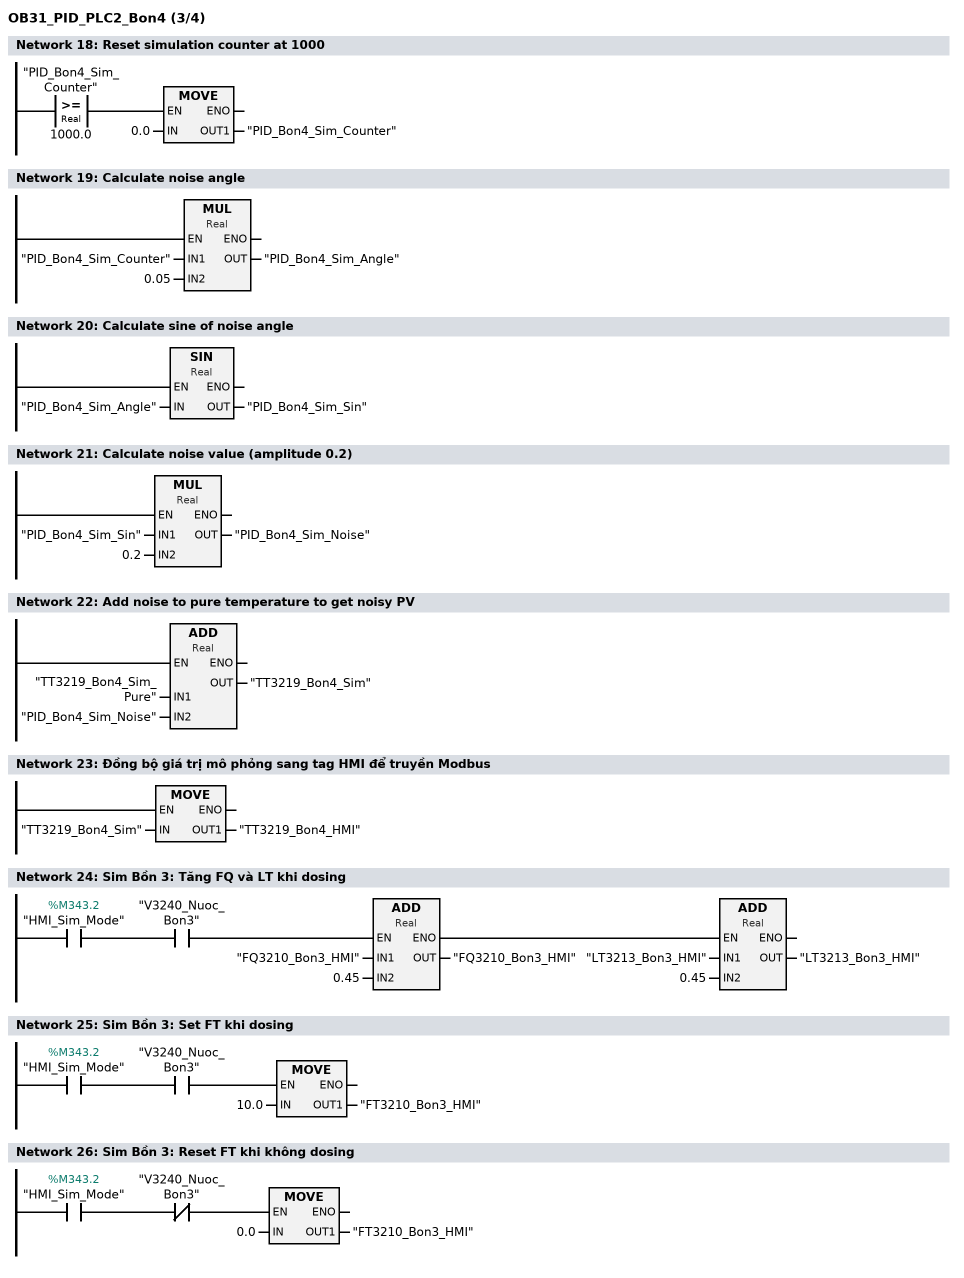
   RUNG wire#powerrail
      { S7_Templates := "SrcType := Real" } GE_Contact(in1 := "PID_Bon4_Sim_Counter", in2 := 1000.0)
      { S7_GenerateENO := "TRUE" } Move(in := 0.0, out1 => "PID_Bon4_Sim_Counter")
   END_RUNG
   // the same network as SCL:
   IF "PID_Bon4_Sim_Counter" >= 1000.0 THEN "PID_Bon4_Sim_Counter" := 0.0; END_IF;
END_REGION

REGION Network 19: Calculate noise angle
   RUNG wire#powerrail
      { S7_Templates := "SrcType := Real"; S7_GenerateENO := "TRUE" } Mul(in1 := "PID_Bon4_Sim_Counter", in2 := 0.05, out => "PID_Bon4_Sim_Angle")
   END_RUNG
   // the same network as SCL:
   "PID_Bon4_Sim_Angle" := "PID_Bon4_Sim_Counter" * 0.05;
END_REGION

REGION Network 20: Calculate sine of noise angle
   "PID_Bon4_Sim_Sin" := SIN("PID_Bon4_Sim_Angle");
END_REGION

REGION Network 21: Calculate noise value (amplitude 0.2)
   RUNG wire#powerrail
      { S7_Templates := "SrcType := Real"; S7_GenerateENO := "TRUE" } Mul(in1 := "PID_Bon4_Sim_Sin", in2 := 0.2, out => "PID_Bon4_Sim_Noise")
   END_RUNG
   // the same network as SCL:
   "PID_Bon4_Sim_Noise" := "PID_Bon4_Sim_Sin" * 0.2;
END_REGION

REGION Network 22: Add noise to pure temperature to get noisy PV
   RUNG wire#powerrail
      { S7_Templates := "SrcType := Real"; S7_GenerateENO := "TRUE" } Add(in1 := "TT3219_Bon4_Sim_Pure", in2 := "PID_Bon4_Sim_Noise", out => "TT3219_Bon4_Sim")
   END_RUNG
   // the same network as SCL:
   "TT3219_Bon4_Sim" := "TT3219_Bon4_Sim_Pure" + "PID_Bon4_Sim_Noise";
END_REGION

REGION Network 23: Đồng bộ giá trị mô phỏng sang tag HMI để truyền Modbus
   RUNG wire#powerrail
      { S7_GenerateENO := "TRUE" } Move(in := "TT3219_Bon4_Sim", out1 => "TT3219_Bon4_HMI")
   END_RUNG
   // the same network as SCL:
   "TT3219_Bon4_HMI" := "TT3219_Bon4_Sim";
END_REGION

REGION Network 24: Sim Bồn 3: Tăng FQ và LT khi dosing
   RUNG wire#powerrail
      Contact( "HMI_Sim_Mode" )
      Contact( "V3240_Nuoc_Bon3" )
      { S7_Templates := "SrcType := Real"; S7_GenerateENO := "TRUE" } Add(in1 := "FQ3210_Bon3_HMI", in2 := 0.45, out => "FQ3210_Bon3_HMI")
      { S7_Templates := "SrcType := Real"; S7_GenerateENO := "TRUE" } Add(in1 := "LT3213_Bon3_HMI", in2 := 0.45, out => "LT3213_Bon3_HMI")
   END_RUNG
   // the same network as SCL:
   // ENO of a box is taken as its EN; it also drops when the box reports an error
   IF "HMI_Sim_Mode" AND "V3240_Nuoc_Bon3" THEN
       "FQ3210_Bon3_HMI" := "FQ3210_Bon3_HMI" + 0.45;
       "LT3213_Bon3_HMI" := "LT3213_Bon3_HMI" + 0.45;
   END_IF;
END_REGION

REGION Network 25: Sim Bồn 3: Set FT khi dosing
   RUNG wire#powerrail
      Contact( "HMI_Sim_Mode" )
      Contact( "V3240_Nuoc_Bon3" )
      { S7_GenerateENO := "TRUE" } Move(in := 10.0, out1 => "FT3210_Bon3_HMI")
   END_RUNG
   // the same network as SCL:
   IF "HMI_Sim_Mode" AND "V3240_Nuoc_Bon3" THEN "FT3210_Bon3_HMI" := 10.0; END_IF;
END_REGION

REGION Network 26: Sim Bồn 3: Reset FT khi không dosing
   RUNG wire#powerrail
      Contact( "HMI_Sim_Mode" )
      I_Contact( "V3240_Nuoc_Bon3" )
      { S7_GenerateENO := "TRUE" } Move(in := 0.0, out1 => "FT3210_Bon3_HMI")
   END_RUNG
   // the same network as SCL:
   IF "HMI_Sim_Mode" AND NOT "V3240_Nuoc_Bon3" THEN "FT3210_Bon3_HMI" := 0.0; END_IF;
END_REGION

REGION Network 27: Sim Bồn 3: Giảm LT khi xả đáy
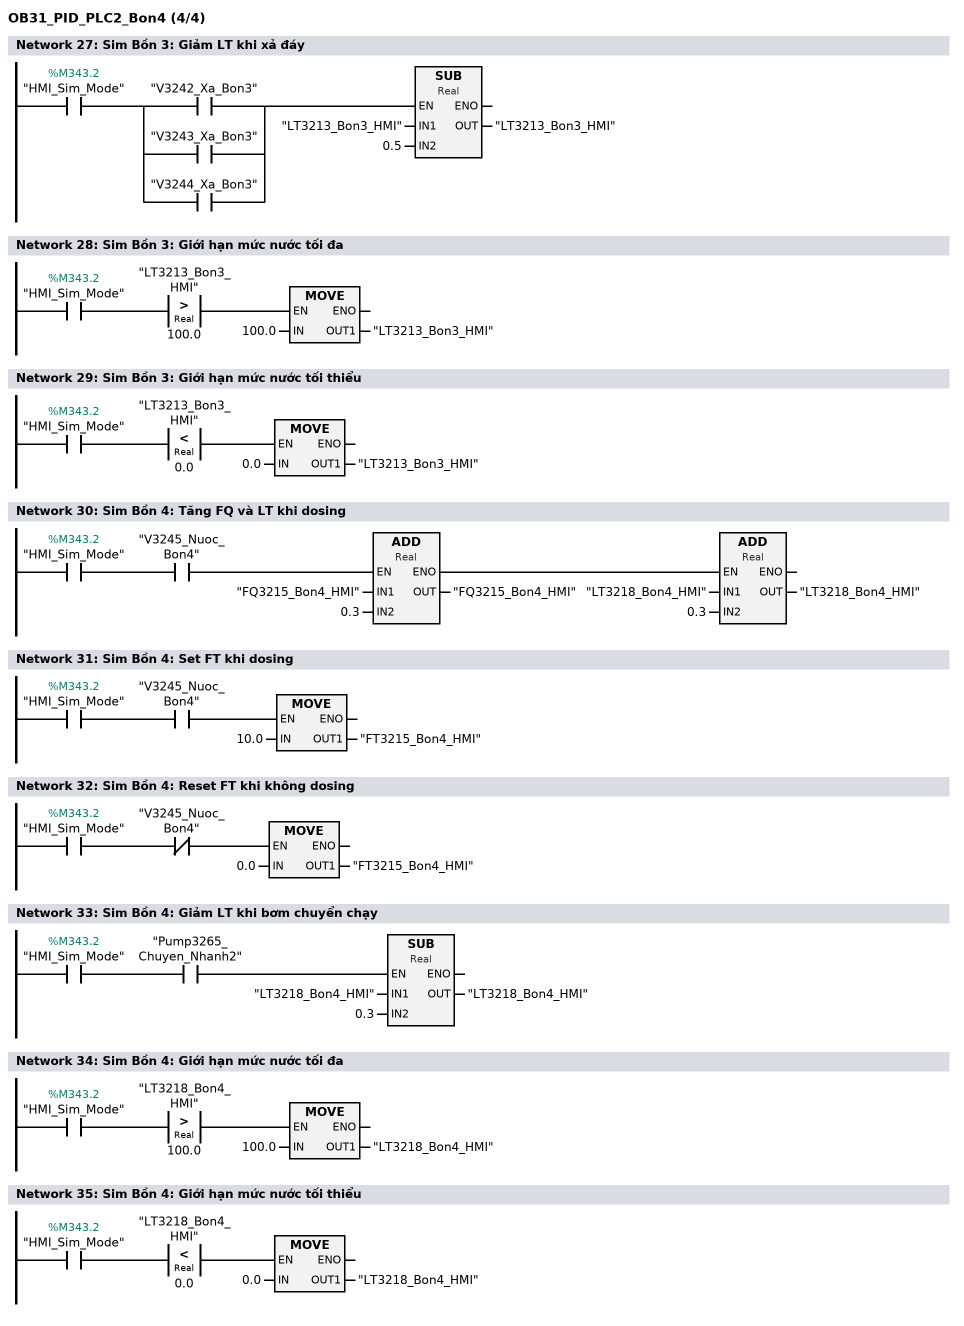
   RUNG wire#powerrail
      Contact( "HMI_Sim_Mode" )
      wire#w1
      Contact( "V3242_Xa_Bon3" )
      wire#w2
      { S7_Templates := "SrcType := Real"; S7_GenerateENO := "TRUE" } Sub(in1 := "LT3213_Bon3_HMI", in2 := 0.5, out => "LT3213_Bon3_HMI")
   END_RUNG
   RUNG wire#w1
      Contact( "V3243_Xa_Bon3" )
   END_RUNG wire#w2
   RUNG wire#w1
      Contact( "V3244_Xa_Bon3" )
   END_RUNG wire#w2
   // the same network as SCL:
   IF "HMI_Sim_Mode" AND ("V3242_Xa_Bon3" OR "V3243_Xa_Bon3" OR "V3244_Xa_Bon3") THEN
       "LT3213_Bon3_HMI" := "LT3213_Bon3_HMI" - 0.5;
   END_IF;
END_REGION

REGION Network 28: Sim Bồn 3: Giới hạn mức nước tối đa
   RUNG wire#powerrail
      Contact( "HMI_Sim_Mode" )
      { S7_Templates := "SrcType := Real" } GT_Contact(in1 := "LT3213_Bon3_HMI", in2 := 100.0)
      { S7_GenerateENO := "TRUE" } Move(in := 100.0, out1 => "LT3213_Bon3_HMI")
   END_RUNG
   // the same network as SCL:
   IF "HMI_Sim_Mode" AND ("LT3213_Bon3_HMI" > 100.0) THEN "LT3213_Bon3_HMI" := 100.0; END_IF;
END_REGION

REGION Network 29: Sim Bồn 3: Giới hạn mức nước tối thiểu
   RUNG wire#powerrail
      Contact( "HMI_Sim_Mode" )
      { S7_Templates := "SrcType := Real" } LT_Contact(in1 := "LT3213_Bon3_HMI", in2 := 0.0)
      { S7_GenerateENO := "TRUE" } Move(in := 0.0, out1 => "LT3213_Bon3_HMI")
   END_RUNG
   // the same network as SCL:
   IF "HMI_Sim_Mode" AND ("LT3213_Bon3_HMI" < 0.0) THEN "LT3213_Bon3_HMI" := 0.0; END_IF;
END_REGION

REGION Network 30: Sim Bồn 4: Tăng FQ và LT khi dosing
   RUNG wire#powerrail
      Contact( "HMI_Sim_Mode" )
      Contact( "V3245_Nuoc_Bon4" )
      { S7_Templates := "SrcType := Real"; S7_GenerateENO := "TRUE" } Add(in1 := "FQ3215_Bon4_HMI", in2 := 0.3, out => "FQ3215_Bon4_HMI")
      { S7_Templates := "SrcType := Real"; S7_GenerateENO := "TRUE" } Add(in1 := "LT3218_Bon4_HMI", in2 := 0.3, out => "LT3218_Bon4_HMI")
   END_RUNG
   // the same network as SCL:
   // ENO of a box is taken as its EN; it also drops when the box reports an error
   IF "HMI_Sim_Mode" AND "V3245_Nuoc_Bon4" THEN
       "FQ3215_Bon4_HMI" := "FQ3215_Bon4_HMI" + 0.3;
       "LT3218_Bon4_HMI" := "LT3218_Bon4_HMI" + 0.3;
   END_IF;
END_REGION

REGION Network 31: Sim Bồn 4: Set FT khi dosing
   RUNG wire#powerrail
      Contact( "HMI_Sim_Mode" )
      Contact( "V3245_Nuoc_Bon4" )
      { S7_GenerateENO := "TRUE" } Move(in := 10.0, out1 => "FT3215_Bon4_HMI")
   END_RUNG
   // the same network as SCL:
   IF "HMI_Sim_Mode" AND "V3245_Nuoc_Bon4" THEN "FT3215_Bon4_HMI" := 10.0; END_IF;
END_REGION

REGION Network 32: Sim Bồn 4: Reset FT khi không dosing
   RUNG wire#powerrail
      Contact( "HMI_Sim_Mode" )
      I_Contact( "V3245_Nuoc_Bon4" )
      { S7_GenerateENO := "TRUE" } Move(in := 0.0, out1 => "FT3215_Bon4_HMI")
   END_RUNG
   // the same network as SCL:
   IF "HMI_Sim_Mode" AND NOT "V3245_Nuoc_Bon4" THEN "FT3215_Bon4_HMI" := 0.0; END_IF;
END_REGION

REGION Network 33: Sim Bồn 4: Giảm LT khi bơm chuyển chạy
   RUNG wire#powerrail
      Contact( "HMI_Sim_Mode" )
      Contact( "Pump3265_Chuyen_Nhanh2" )
      { S7_Templates := "SrcType := Real"; S7_GenerateENO := "TRUE" } Sub(in1 := "LT3218_Bon4_HMI", in2 := 0.3, out => "LT3218_Bon4_HMI")
   END_RUNG
   // the same network as SCL:
   IF "HMI_Sim_Mode" AND "Pump3265_Chuyen_Nhanh2" THEN "LT3218_Bon4_HMI" := "LT3218_Bon4_HMI" - 0.3; END_IF;
END_REGION

REGION Network 34: Sim Bồn 4: Giới hạn mức nước tối đa
   RUNG wire#powerrail
      Contact( "HMI_Sim_Mode" )
      { S7_Templates := "SrcType := Real" } GT_Contact(in1 := "LT3218_Bon4_HMI", in2 := 100.0)
      { S7_GenerateENO := "TRUE" } Move(in := 100.0, out1 => "LT3218_Bon4_HMI")
   END_RUNG
   // the same network as SCL:
   IF "HMI_Sim_Mode" AND ("LT3218_Bon4_HMI" > 100.0) THEN "LT3218_Bon4_HMI" := 100.0; END_IF;
END_REGION

REGION Network 35: Sim Bồn 4: Giới hạn mức nước tối thiểu
   RUNG wire#powerrail
      Contact( "HMI_Sim_Mode" )
      { S7_Templates := "SrcType := Real" } LT_Contact(in1 := "LT3218_Bon4_HMI", in2 := 0.0)
      { S7_GenerateENO := "TRUE" } Move(in := 0.0, out1 => "LT3218_Bon4_HMI")
   END_RUNG
   // the same network as SCL:
   IF "HMI_Sim_Mode" AND ("LT3218_Bon4_HMI" < 0.0) THEN "LT3218_Bon4_HMI" := 0.0; END_IF;
END_REGION
END_ORGANIZATION_BLOCK

FUNCTION "FC_HMI_Mirror_PLC2" : Void   // FC41, LAD
{ S7_Optimized_Access := 'TRUE' }
VERSION : 0.1
// stored: AutoNumber true, IsIECCheckEnabled false, SetENOAutomatically false, UDAEnableTagReadback false
BEGIN

REGION Network 1: Mirror V3240_Nuoc_Bon3
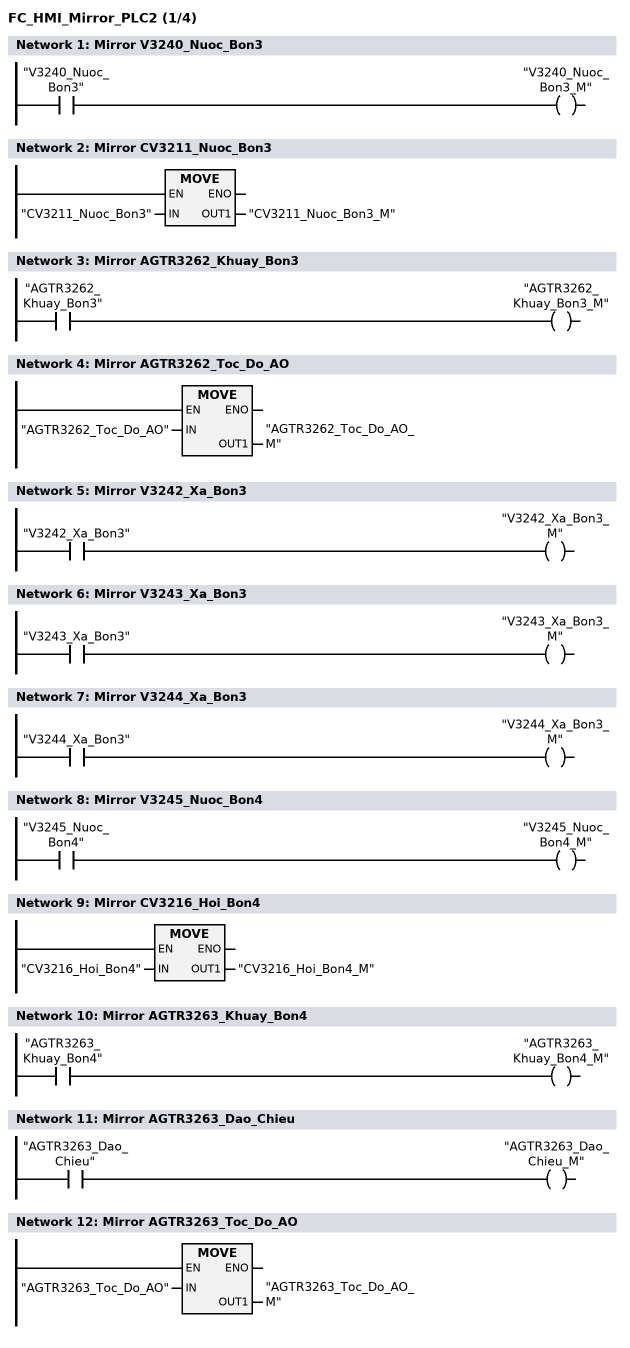
   RUNG wire#powerrail
      Contact( "V3240_Nuoc_Bon3" )
      Coil( "V3240_Nuoc_Bon3_M" )
   END_RUNG
   // the same network as SCL:
   "V3240_Nuoc_Bon3_M" := "V3240_Nuoc_Bon3";
END_REGION

REGION Network 2: Mirror CV3211_Nuoc_Bon3
   RUNG wire#powerrail
      { S7_GenerateENO := "TRUE" } Move(in := "CV3211_Nuoc_Bon3", out1 => "CV3211_Nuoc_Bon3_M")
   END_RUNG
   // the same network as SCL:
   "CV3211_Nuoc_Bon3_M" := "CV3211_Nuoc_Bon3";
END_REGION

REGION Network 3: Mirror AGTR3262_Khuay_Bon3
   RUNG wire#powerrail
      Contact( "AGTR3262_Khuay_Bon3" )
      Coil( "AGTR3262_Khuay_Bon3_M" )
   END_RUNG
   // the same network as SCL:
   "AGTR3262_Khuay_Bon3_M" := "AGTR3262_Khuay_Bon3";
END_REGION

REGION Network 4: Mirror AGTR3262_Toc_Do_AO
   RUNG wire#powerrail
      { S7_GenerateENO := "TRUE" } Move(in := "AGTR3262_Toc_Do_AO", out1 => "AGTR3262_Toc_Do_AO_M")
   END_RUNG
   // the same network as SCL:
   "AGTR3262_Toc_Do_AO_M" := "AGTR3262_Toc_Do_AO";
END_REGION

REGION Network 5: Mirror V3242_Xa_Bon3
   RUNG wire#powerrail
      Contact( "V3242_Xa_Bon3" )
      Coil( "V3242_Xa_Bon3_M" )
   END_RUNG
   // the same network as SCL:
   "V3242_Xa_Bon3_M" := "V3242_Xa_Bon3";
END_REGION

REGION Network 6: Mirror V3243_Xa_Bon3
   RUNG wire#powerrail
      Contact( "V3243_Xa_Bon3" )
      Coil( "V3243_Xa_Bon3_M" )
   END_RUNG
   // the same network as SCL:
   "V3243_Xa_Bon3_M" := "V3243_Xa_Bon3";
END_REGION

REGION Network 7: Mirror V3244_Xa_Bon3
   RUNG wire#powerrail
      Contact( "V3244_Xa_Bon3" )
      Coil( "V3244_Xa_Bon3_M" )
   END_RUNG
   // the same network as SCL:
   "V3244_Xa_Bon3_M" := "V3244_Xa_Bon3";
END_REGION

REGION Network 8: Mirror V3245_Nuoc_Bon4
   RUNG wire#powerrail
      Contact( "V3245_Nuoc_Bon4" )
      Coil( "V3245_Nuoc_Bon4_M" )
   END_RUNG
   // the same network as SCL:
   "V3245_Nuoc_Bon4_M" := "V3245_Nuoc_Bon4";
END_REGION

REGION Network 9: Mirror CV3216_Hoi_Bon4
   RUNG wire#powerrail
      { S7_GenerateENO := "TRUE" } Move(in := "CV3216_Hoi_Bon4", out1 => "CV3216_Hoi_Bon4_M")
   END_RUNG
   // the same network as SCL:
   "CV3216_Hoi_Bon4_M" := "CV3216_Hoi_Bon4";
END_REGION

REGION Network 10: Mirror AGTR3263_Khuay_Bon4
   RUNG wire#powerrail
      Contact( "AGTR3263_Khuay_Bon4" )
      Coil( "AGTR3263_Khuay_Bon4_M" )
   END_RUNG
   // the same network as SCL:
   "AGTR3263_Khuay_Bon4_M" := "AGTR3263_Khuay_Bon4";
END_REGION

REGION Network 11: Mirror AGTR3263_Dao_Chieu
   RUNG wire#powerrail
      Contact( "AGTR3263_Dao_Chieu" )
      Coil( "AGTR3263_Dao_Chieu_M" )
   END_RUNG
   // the same network as SCL:
   "AGTR3263_Dao_Chieu_M" := "AGTR3263_Dao_Chieu";
END_REGION

REGION Network 12: Mirror AGTR3263_Toc_Do_AO
   RUNG wire#powerrail
      { S7_GenerateENO := "TRUE" } Move(in := "AGTR3263_Toc_Do_AO", out1 => "AGTR3263_Toc_Do_AO_M")
   END_RUNG
   // the same network as SCL:
   "AGTR3263_Toc_Do_AO_M" := "AGTR3263_Toc_Do_AO";
END_REGION

REGION Network 13: Mirror V3247_Xa_Bon4
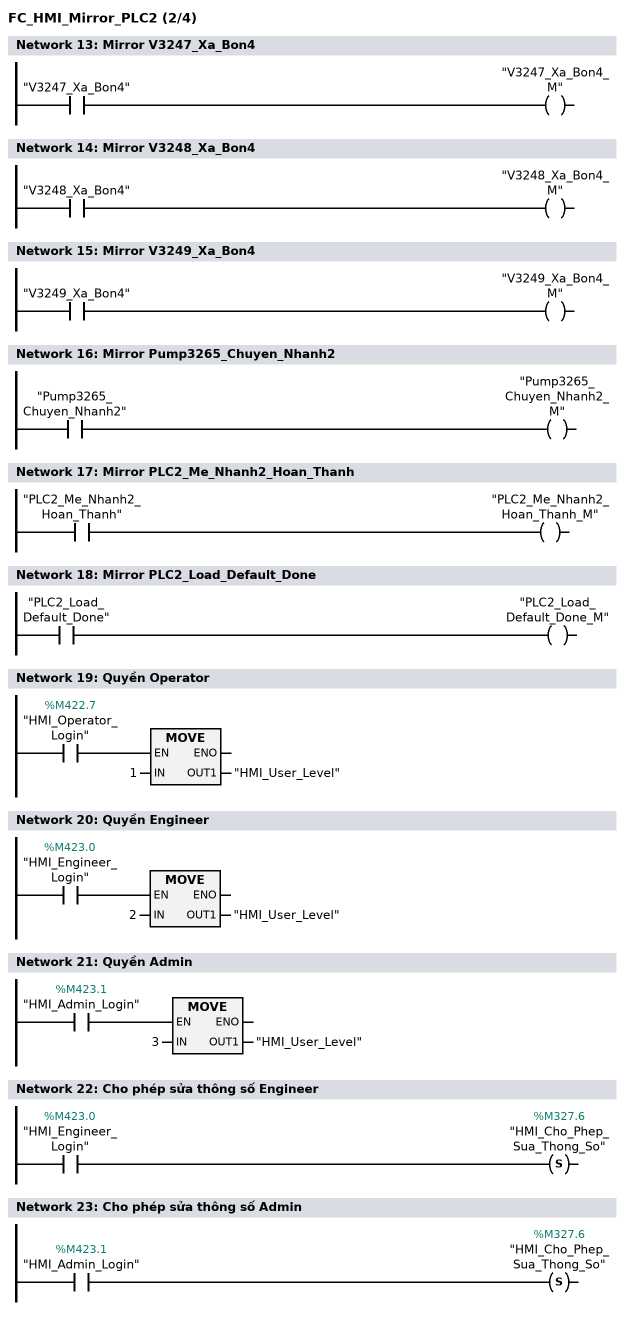
   RUNG wire#powerrail
      Contact( "V3247_Xa_Bon4" )
      Coil( "V3247_Xa_Bon4_M" )
   END_RUNG
   // the same network as SCL:
   "V3247_Xa_Bon4_M" := "V3247_Xa_Bon4";
END_REGION

REGION Network 14: Mirror V3248_Xa_Bon4
   RUNG wire#powerrail
      Contact( "V3248_Xa_Bon4" )
      Coil( "V3248_Xa_Bon4_M" )
   END_RUNG
   // the same network as SCL:
   "V3248_Xa_Bon4_M" := "V3248_Xa_Bon4";
END_REGION

REGION Network 15: Mirror V3249_Xa_Bon4
   RUNG wire#powerrail
      Contact( "V3249_Xa_Bon4" )
      Coil( "V3249_Xa_Bon4_M" )
   END_RUNG
   // the same network as SCL:
   "V3249_Xa_Bon4_M" := "V3249_Xa_Bon4";
END_REGION

REGION Network 16: Mirror Pump3265_Chuyen_Nhanh2
   RUNG wire#powerrail
      Contact( "Pump3265_Chuyen_Nhanh2" )
      Coil( "Pump3265_Chuyen_Nhanh2_M" )
   END_RUNG
   // the same network as SCL:
   "Pump3265_Chuyen_Nhanh2_M" := "Pump3265_Chuyen_Nhanh2";
END_REGION

REGION Network 17: Mirror PLC2_Me_Nhanh2_Hoan_Thanh
   RUNG wire#powerrail
      Contact( "PLC2_Me_Nhanh2_Hoan_Thanh" )
      Coil( "PLC2_Me_Nhanh2_Hoan_Thanh_M" )
   END_RUNG
   // the same network as SCL:
   "PLC2_Me_Nhanh2_Hoan_Thanh_M" := "PLC2_Me_Nhanh2_Hoan_Thanh";
END_REGION

REGION Network 18: Mirror PLC2_Load_Default_Done
   RUNG wire#powerrail
      Contact( "PLC2_Load_Default_Done" )
      Coil( "PLC2_Load_Default_Done_M" )
   END_RUNG
   // the same network as SCL:
   "PLC2_Load_Default_Done_M" := "PLC2_Load_Default_Done";
END_REGION

REGION Network 19: Quyền Operator
   RUNG wire#powerrail
      Contact( "HMI_Operator_Login" )
      { S7_GenerateENO := "TRUE" } Move(in := 1, out1 => "HMI_User_Level")
   END_RUNG
   // the same network as SCL:
   IF "HMI_Operator_Login" THEN "HMI_User_Level" := 1; END_IF;
END_REGION

REGION Network 20: Quyền Engineer
   RUNG wire#powerrail
      Contact( "HMI_Engineer_Login" )
      { S7_GenerateENO := "TRUE" } Move(in := 2, out1 => "HMI_User_Level")
   END_RUNG
   // the same network as SCL:
   IF "HMI_Engineer_Login" THEN "HMI_User_Level" := 2; END_IF;
END_REGION

REGION Network 21: Quyền Admin
   RUNG wire#powerrail
      Contact( "HMI_Admin_Login" )
      { S7_GenerateENO := "TRUE" } Move(in := 3, out1 => "HMI_User_Level")
   END_RUNG
   // the same network as SCL:
   IF "HMI_Admin_Login" THEN "HMI_User_Level" := 3; END_IF;
END_REGION

REGION Network 22: Cho phép sửa thông số Engineer
   RUNG wire#powerrail
      Contact( "HMI_Engineer_Login" )
      S_Coil( "HMI_Cho_Phep_Sua_Thong_So" )
   END_RUNG
   // the same network as SCL:
   IF "HMI_Engineer_Login" THEN "HMI_Cho_Phep_Sua_Thong_So" := TRUE; END_IF;
END_REGION

REGION Network 23: Cho phép sửa thông số Admin
   RUNG wire#powerrail
      Contact( "HMI_Admin_Login" )
      S_Coil( "HMI_Cho_Phep_Sua_Thong_So" )
   END_RUNG
   // the same network as SCL:
   IF "HMI_Admin_Login" THEN "HMI_Cho_Phep_Sua_Thong_So" := TRUE; END_IF;
END_REGION

REGION Network 24: Operator không được sửa thông số
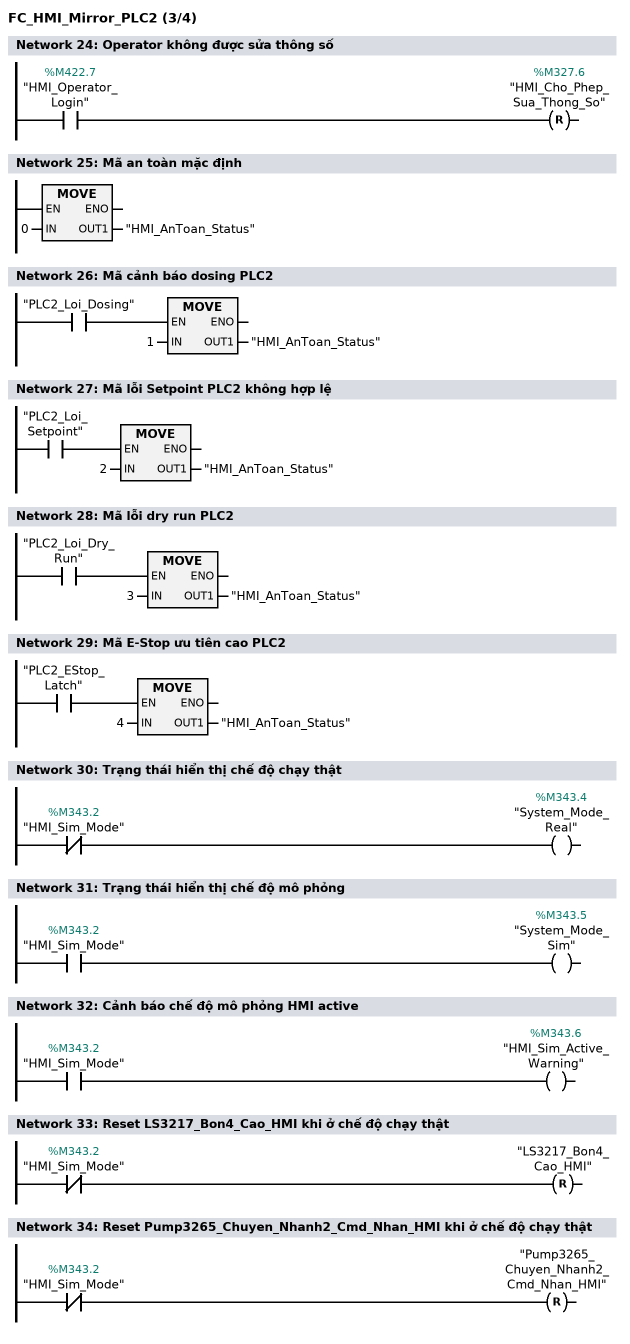
   RUNG wire#powerrail
      Contact( "HMI_Operator_Login" )
      R_Coil( "HMI_Cho_Phep_Sua_Thong_So" )
   END_RUNG
   // the same network as SCL:
   IF "HMI_Operator_Login" THEN "HMI_Cho_Phep_Sua_Thong_So" := FALSE; END_IF;
END_REGION

REGION Network 25: Mã an toàn mặc định
   RUNG wire#powerrail
      { S7_GenerateENO := "TRUE" } Move(in := 0, out1 => "HMI_AnToan_Status")
   END_RUNG
   // the same network as SCL:
   "HMI_AnToan_Status" := 0;
END_REGION

REGION Network 26: Mã cảnh báo dosing PLC2
   RUNG wire#powerrail
      Contact( "PLC2_Loi_Dosing" )
      { S7_GenerateENO := "TRUE" } Move(in := 1, out1 => "HMI_AnToan_Status")
   END_RUNG
   // the same network as SCL:
   IF "PLC2_Loi_Dosing" THEN "HMI_AnToan_Status" := 1; END_IF;
END_REGION

REGION Network 27: Mã lỗi Setpoint PLC2 không hợp lệ
   RUNG wire#powerrail
      Contact( "PLC2_Loi_Setpoint" )
      { S7_GenerateENO := "TRUE" } Move(in := 2, out1 => "HMI_AnToan_Status")
   END_RUNG
   // the same network as SCL:
   IF "PLC2_Loi_Setpoint" THEN "HMI_AnToan_Status" := 2; END_IF;
END_REGION

REGION Network 28: Mã lỗi dry run PLC2
   RUNG wire#powerrail
      Contact( "PLC2_Loi_Dry_Run" )
      { S7_GenerateENO := "TRUE" } Move(in := 3, out1 => "HMI_AnToan_Status")
   END_RUNG
   // the same network as SCL:
   IF "PLC2_Loi_Dry_Run" THEN "HMI_AnToan_Status" := 3; END_IF;
END_REGION

REGION Network 29: Mã E-Stop ưu tiên cao PLC2
   RUNG wire#powerrail
      Contact( "PLC2_EStop_Latch" )
      { S7_GenerateENO := "TRUE" } Move(in := 4, out1 => "HMI_AnToan_Status")
   END_RUNG
   // the same network as SCL:
   IF "PLC2_EStop_Latch" THEN "HMI_AnToan_Status" := 4; END_IF;
END_REGION

REGION Network 30: Trạng thái hiển thị chế độ chạy thật
   RUNG wire#powerrail
      I_Contact( "HMI_Sim_Mode" )
      Coil( "System_Mode_Real" )
   END_RUNG
   // the same network as SCL:
   "System_Mode_Real" := NOT "HMI_Sim_Mode";
END_REGION

REGION Network 31: Trạng thái hiển thị chế độ mô phỏng
   RUNG wire#powerrail
      Contact( "HMI_Sim_Mode" )
      Coil( "System_Mode_Sim" )
   END_RUNG
   // the same network as SCL:
   "System_Mode_Sim" := "HMI_Sim_Mode";
END_REGION

REGION Network 32: Cảnh báo chế độ mô phỏng HMI active
   RUNG wire#powerrail
      Contact( "HMI_Sim_Mode" )
      Coil( "HMI_Sim_Active_Warning" )
   END_RUNG
   // the same network as SCL:
   "HMI_Sim_Active_Warning" := "HMI_Sim_Mode";
END_REGION

REGION Network 33: Reset LS3217_Bon4_Cao_HMI khi ở chế độ chạy thật
   RUNG wire#powerrail
      I_Contact( "HMI_Sim_Mode" )
      R_Coil( "LS3217_Bon4_Cao_HMI" )
   END_RUNG
   // the same network as SCL:
   IF NOT "HMI_Sim_Mode" THEN "LS3217_Bon4_Cao_HMI" := FALSE; END_IF;
END_REGION

REGION Network 34: Reset Pump3265_Chuyen_Nhanh2_Cmd_Nhan_HMI khi ở chế độ chạy thật
   RUNG wire#powerrail
      I_Contact( "HMI_Sim_Mode" )
      R_Coil( "Pump3265_Chuyen_Nhanh2_Cmd_Nhan_HMI" )
   END_RUNG
   // the same network as SCL:
   IF NOT "HMI_Sim_Mode" THEN "Pump3265_Chuyen_Nhanh2_Cmd_Nhan_HMI" := FALSE; END_IF;
END_REGION

REGION Network 35: Reset PLC2_Load_Default_Cmd_Nhan_HMI khi ở chế độ chạy thật
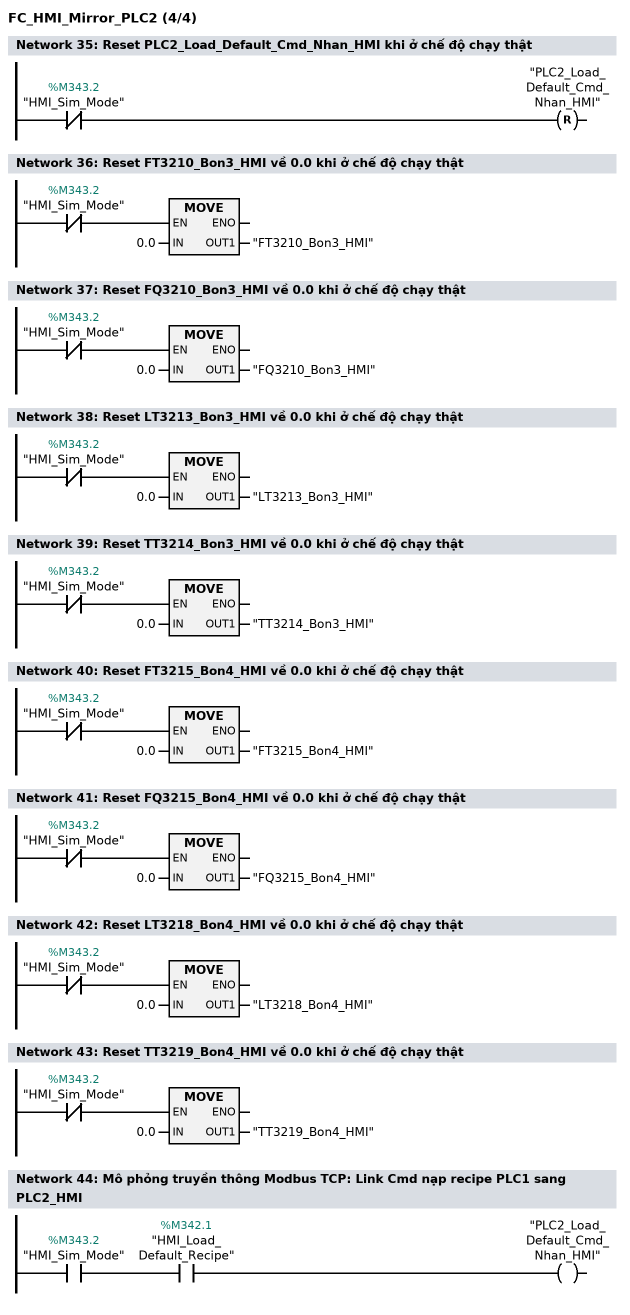
   RUNG wire#powerrail
      I_Contact( "HMI_Sim_Mode" )
      R_Coil( "PLC2_Load_Default_Cmd_Nhan_HMI" )
   END_RUNG
   // the same network as SCL:
   IF NOT "HMI_Sim_Mode" THEN "PLC2_Load_Default_Cmd_Nhan_HMI" := FALSE; END_IF;
END_REGION

REGION Network 36: Reset FT3210_Bon3_HMI về 0.0 khi ở chế độ chạy thật
   RUNG wire#powerrail
      I_Contact( "HMI_Sim_Mode" )
      { S7_GenerateENO := "TRUE" } Move(in := 0.0, out1 => "FT3210_Bon3_HMI")
   END_RUNG
   // the same network as SCL:
   IF NOT "HMI_Sim_Mode" THEN "FT3210_Bon3_HMI" := 0.0; END_IF;
END_REGION

REGION Network 37: Reset FQ3210_Bon3_HMI về 0.0 khi ở chế độ chạy thật
   RUNG wire#powerrail
      I_Contact( "HMI_Sim_Mode" )
      { S7_GenerateENO := "TRUE" } Move(in := 0.0, out1 => "FQ3210_Bon3_HMI")
   END_RUNG
   // the same network as SCL:
   IF NOT "HMI_Sim_Mode" THEN "FQ3210_Bon3_HMI" := 0.0; END_IF;
END_REGION

REGION Network 38: Reset LT3213_Bon3_HMI về 0.0 khi ở chế độ chạy thật
   RUNG wire#powerrail
      I_Contact( "HMI_Sim_Mode" )
      { S7_GenerateENO := "TRUE" } Move(in := 0.0, out1 => "LT3213_Bon3_HMI")
   END_RUNG
   // the same network as SCL:
   IF NOT "HMI_Sim_Mode" THEN "LT3213_Bon3_HMI" := 0.0; END_IF;
END_REGION

REGION Network 39: Reset TT3214_Bon3_HMI về 0.0 khi ở chế độ chạy thật
   RUNG wire#powerrail
      I_Contact( "HMI_Sim_Mode" )
      { S7_GenerateENO := "TRUE" } Move(in := 0.0, out1 => "TT3214_Bon3_HMI")
   END_RUNG
   // the same network as SCL:
   IF NOT "HMI_Sim_Mode" THEN "TT3214_Bon3_HMI" := 0.0; END_IF;
END_REGION

REGION Network 40: Reset FT3215_Bon4_HMI về 0.0 khi ở chế độ chạy thật
   RUNG wire#powerrail
      I_Contact( "HMI_Sim_Mode" )
      { S7_GenerateENO := "TRUE" } Move(in := 0.0, out1 => "FT3215_Bon4_HMI")
   END_RUNG
   // the same network as SCL:
   IF NOT "HMI_Sim_Mode" THEN "FT3215_Bon4_HMI" := 0.0; END_IF;
END_REGION

REGION Network 41: Reset FQ3215_Bon4_HMI về 0.0 khi ở chế độ chạy thật
   RUNG wire#powerrail
      I_Contact( "HMI_Sim_Mode" )
      { S7_GenerateENO := "TRUE" } Move(in := 0.0, out1 => "FQ3215_Bon4_HMI")
   END_RUNG
   // the same network as SCL:
   IF NOT "HMI_Sim_Mode" THEN "FQ3215_Bon4_HMI" := 0.0; END_IF;
END_REGION

REGION Network 42: Reset LT3218_Bon4_HMI về 0.0 khi ở chế độ chạy thật
   RUNG wire#powerrail
      I_Contact( "HMI_Sim_Mode" )
      { S7_GenerateENO := "TRUE" } Move(in := 0.0, out1 => "LT3218_Bon4_HMI")
   END_RUNG
   // the same network as SCL:
   IF NOT "HMI_Sim_Mode" THEN "LT3218_Bon4_HMI" := 0.0; END_IF;
END_REGION

REGION Network 43: Reset TT3219_Bon4_HMI về 0.0 khi ở chế độ chạy thật
   RUNG wire#powerrail
      I_Contact( "HMI_Sim_Mode" )
      { S7_GenerateENO := "TRUE" } Move(in := 0.0, out1 => "TT3219_Bon4_HMI")
   END_RUNG
   // the same network as SCL:
   IF NOT "HMI_Sim_Mode" THEN "TT3219_Bon4_HMI" := 0.0; END_IF;
END_REGION

REGION Network 44: Mô phỏng truyền thông Modbus TCP: Link Cmd nạp recipe PLC1 sang PLC2_HMI
   RUNG wire#powerrail
      Contact( "HMI_Sim_Mode" )
      Contact( "HMI_Load_Default_Recipe" )
      Coil( "PLC2_Load_Default_Cmd_Nhan_HMI" )
   END_RUNG
   // the same network as SCL:
   "PLC2_Load_Default_Cmd_Nhan_HMI" := "HMI_Sim_Mode" AND "HMI_Load_Default_Recipe";
END_REGION
END_FUNCTION

FUNCTION "FC_Init_Default_Recipe_PLC2" : Void   // FC51, LAD
{ S7_Optimized_Access := 'TRUE' }
VERSION : 0.1
// stored: AutoNumber true, IsIECCheckEnabled false, SetENOAutomatically false, UDAEnableTagReadback false
BEGIN

REGION Network 1: Kích hoạt nạp recipe mặc định lần đầu scan PLC2
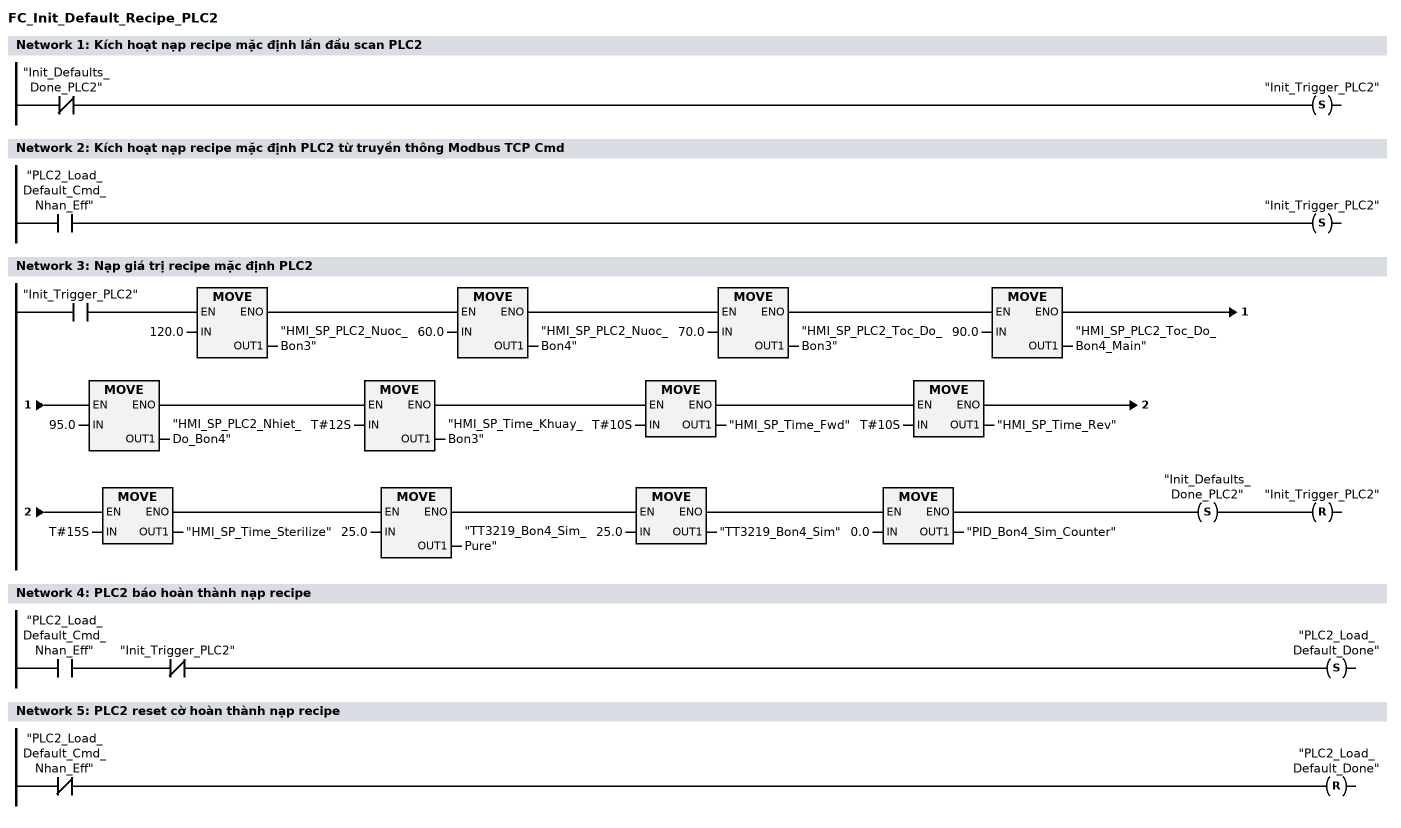
   RUNG wire#powerrail
      I_Contact( "Init_Defaults_Done_PLC2" )
      S_Coil( "Init_Trigger_PLC2" )
   END_RUNG
   // the same network as SCL:
   IF NOT "Init_Defaults_Done_PLC2" THEN "Init_Trigger_PLC2" := TRUE; END_IF;
END_REGION

REGION Network 2: Kích hoạt nạp recipe mặc định PLC2 từ truyền thông Modbus TCP Cmd
   RUNG wire#powerrail
      Contact( "PLC2_Load_Default_Cmd_Nhan_Eff" )
      S_Coil( "Init_Trigger_PLC2" )
   END_RUNG
   // the same network as SCL:
   IF "PLC2_Load_Default_Cmd_Nhan_Eff" THEN "Init_Trigger_PLC2" := TRUE; END_IF;
END_REGION

REGION Network 3: Nạp giá trị recipe mặc định PLC2
   RUNG wire#powerrail
      Contact( "Init_Trigger_PLC2" )
      { S7_GenerateENO := "TRUE" } Move(in := 120.0, out1 => "HMI_SP_PLC2_Nuoc_Bon3")
      { S7_GenerateENO := "TRUE" } Move(in := 60.0, out1 => "HMI_SP_PLC2_Nuoc_Bon4")
      { S7_GenerateENO := "TRUE" } Move(in := 70.0, out1 => "HMI_SP_PLC2_Toc_Do_Bon3")
      { S7_GenerateENO := "TRUE" } Move(in := 90.0, out1 => "HMI_SP_PLC2_Toc_Do_Bon4_Main")
      { S7_GenerateENO := "TRUE" } Move(in := 95.0, out1 => "HMI_SP_PLC2_Nhiet_Do_Bon4")
      { S7_GenerateENO := "TRUE" } Move(in := T#12S, out1 => "HMI_SP_Time_Khuay_Bon3")
      { S7_GenerateENO := "TRUE" } Move(in := T#10S, out1 => "HMI_SP_Time_Fwd")
      { S7_GenerateENO := "TRUE" } Move(in := T#10S, out1 => "HMI_SP_Time_Rev")
      { S7_GenerateENO := "TRUE" } Move(in := T#15S, out1 => "HMI_SP_Time_Sterilize")
      { S7_GenerateENO := "TRUE" } Move(in := 25.0, out1 => "TT3219_Bon4_Sim_Pure")
      { S7_GenerateENO := "TRUE" } Move(in := 25.0, out1 => "TT3219_Bon4_Sim")
      { S7_GenerateENO := "TRUE" } Move(in := 0.0, out1 => "PID_Bon4_Sim_Counter")
      S_Coil( "Init_Defaults_Done_PLC2" )
      R_Coil( "Init_Trigger_PLC2" )
   END_RUNG
   // the same network as SCL:
   // ENO of a box is taken as its EN; it also drops when the box reports an error
   IF "Init_Trigger_PLC2" THEN
       "HMI_SP_PLC2_Nuoc_Bon3" := 120.0;
       "HMI_SP_PLC2_Nuoc_Bon4" := 60.0;
       "HMI_SP_PLC2_Toc_Do_Bon3" := 70.0;
       "HMI_SP_PLC2_Toc_Do_Bon4_Main" := 90.0;
       "HMI_SP_PLC2_Nhiet_Do_Bon4" := 95.0;
       "HMI_SP_Time_Khuay_Bon3" := T#12S;
       "HMI_SP_Time_Fwd" := T#10S;
       "HMI_SP_Time_Rev" := T#10S;
       "HMI_SP_Time_Sterilize" := T#15S;
       "TT3219_Bon4_Sim_Pure" := 25.0;
       "TT3219_Bon4_Sim" := 25.0;
       "PID_Bon4_Sim_Counter" := 0.0;
       "Init_Defaults_Done_PLC2" := TRUE;
       "Init_Trigger_PLC2" := FALSE;
   END_IF;
END_REGION

REGION Network 4: PLC2 báo hoàn thành nạp recipe
   RUNG wire#powerrail
      Contact( "PLC2_Load_Default_Cmd_Nhan_Eff" )
      I_Contact( "Init_Trigger_PLC2" )
      S_Coil( "PLC2_Load_Default_Done" )
   END_RUNG
   // the same network as SCL:
   IF "PLC2_Load_Default_Cmd_Nhan_Eff" AND NOT "Init_Trigger_PLC2" THEN
       "PLC2_Load_Default_Done" := TRUE;
   END_IF;
END_REGION

REGION Network 5: PLC2 reset cờ hoàn thành nạp recipe
   RUNG wire#powerrail
      I_Contact( "PLC2_Load_Default_Cmd_Nhan_Eff" )
      R_Coil( "PLC2_Load_Default_Done" )
   END_RUNG
   // the same network as SCL:
   IF NOT "PLC2_Load_Default_Cmd_Nhan_Eff" THEN "PLC2_Load_Default_Done" := FALSE; END_IF;
END_REGION
END_FUNCTION

FUNCTION "FC_PLC2_Mixing" : Void   // FC20, LAD
{ S7_Optimized_Access := 'TRUE' }
VERSION : 0.1
// stored: AutoNumber true, IsIECCheckEnabled false, SetENOAutomatically false, UDAEnableTagReadback false
   VAR_TEMP   // added for the SCL form of the ladder/FBD networks
      _w1 : Bool;
   END_VAR
BEGIN

REGION Network 1: Khóa nút nhấn Start HMI qua Run Enable PLC2
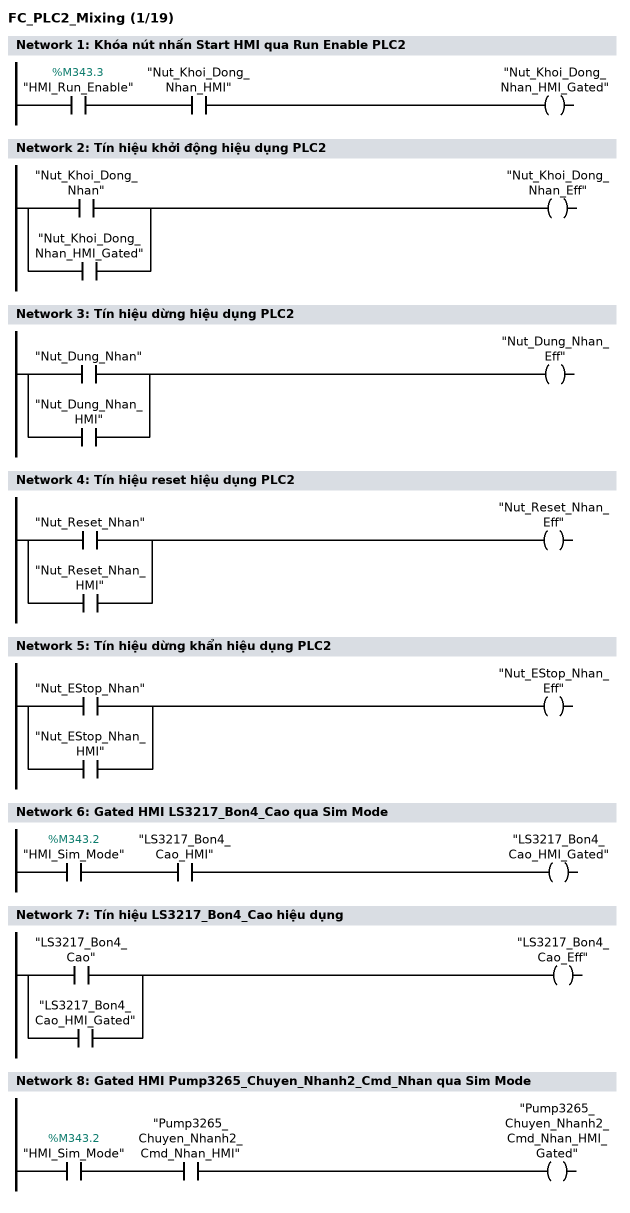
   RUNG wire#powerrail
      Contact( "HMI_Run_Enable" )
      Contact( "Nut_Khoi_Dong_Nhan_HMI" )
      Coil( "Nut_Khoi_Dong_Nhan_HMI_Gated" )
   END_RUNG
   // the same network as SCL:
   "Nut_Khoi_Dong_Nhan_HMI_Gated" := "HMI_Run_Enable" AND "Nut_Khoi_Dong_Nhan_HMI";
END_REGION

REGION Network 2: Tín hiệu khởi động hiệu dụng PLC2
   RUNG wire#powerrail
      Contact( "Nut_Khoi_Dong_Nhan" )
      wire#w1
      Coil( "Nut_Khoi_Dong_Nhan_Eff" )
   END_RUNG
   RUNG wire#powerrail
      Contact( "Nut_Khoi_Dong_Nhan_HMI_Gated" )
   END_RUNG wire#w1
   // the same network as SCL:
   "Nut_Khoi_Dong_Nhan_Eff" := "Nut_Khoi_Dong_Nhan" OR "Nut_Khoi_Dong_Nhan_HMI_Gated";
END_REGION

REGION Network 3: Tín hiệu dừng hiệu dụng PLC2
   RUNG wire#powerrail
      Contact( "Nut_Dung_Nhan" )
      wire#w1
      Coil( "Nut_Dung_Nhan_Eff" )
   END_RUNG
   RUNG wire#powerrail
      Contact( "Nut_Dung_Nhan_HMI" )
   END_RUNG wire#w1
   // the same network as SCL:
   "Nut_Dung_Nhan_Eff" := "Nut_Dung_Nhan" OR "Nut_Dung_Nhan_HMI";
END_REGION

REGION Network 4: Tín hiệu reset hiệu dụng PLC2
   RUNG wire#powerrail
      Contact( "Nut_Reset_Nhan" )
      wire#w1
      Coil( "Nut_Reset_Nhan_Eff" )
   END_RUNG
   RUNG wire#powerrail
      Contact( "Nut_Reset_Nhan_HMI" )
   END_RUNG wire#w1
   // the same network as SCL:
   "Nut_Reset_Nhan_Eff" := "Nut_Reset_Nhan" OR "Nut_Reset_Nhan_HMI";
END_REGION

REGION Network 5: Tín hiệu dừng khẩn hiệu dụng PLC2
   RUNG wire#powerrail
      Contact( "Nut_EStop_Nhan" )
      wire#w1
      Coil( "Nut_EStop_Nhan_Eff" )
   END_RUNG
   RUNG wire#powerrail
      Contact( "Nut_EStop_Nhan_HMI" )
   END_RUNG wire#w1
   // the same network as SCL:
   "Nut_EStop_Nhan_Eff" := "Nut_EStop_Nhan" OR "Nut_EStop_Nhan_HMI";
END_REGION

REGION Network 6: Gated HMI LS3217_Bon4_Cao qua Sim Mode
   RUNG wire#powerrail
      Contact( "HMI_Sim_Mode" )
      Contact( "LS3217_Bon4_Cao_HMI" )
      Coil( "LS3217_Bon4_Cao_HMI_Gated" )
   END_RUNG
   // the same network as SCL:
   "LS3217_Bon4_Cao_HMI_Gated" := "HMI_Sim_Mode" AND "LS3217_Bon4_Cao_HMI";
END_REGION

REGION Network 7: Tín hiệu LS3217_Bon4_Cao hiệu dụng
   RUNG wire#powerrail
      Contact( "LS3217_Bon4_Cao" )
      wire#w1
      Coil( "LS3217_Bon4_Cao_Eff" )
   END_RUNG
   RUNG wire#powerrail
      Contact( "LS3217_Bon4_Cao_HMI_Gated" )
   END_RUNG wire#w1
   // the same network as SCL:
   "LS3217_Bon4_Cao_Eff" := "LS3217_Bon4_Cao" OR "LS3217_Bon4_Cao_HMI_Gated";
END_REGION

REGION Network 8: Gated HMI Pump3265_Chuyen_Nhanh2_Cmd_Nhan qua Sim Mode
   RUNG wire#powerrail
      Contact( "HMI_Sim_Mode" )
      Contact( "Pump3265_Chuyen_Nhanh2_Cmd_Nhan_HMI" )
      Coil( "Pump3265_Chuyen_Nhanh2_Cmd_Nhan_HMI_Gated" )
   END_RUNG
   // the same network as SCL:
   "Pump3265_Chuyen_Nhanh2_Cmd_Nhan_HMI_Gated" := "HMI_Sim_Mode" AND "Pump3265_Chuyen_Nhanh2_Cmd_Nhan_HMI";
END_REGION

REGION Network 9: Tín hiệu Pump3265_Chuyen_Nhanh2_Cmd_Nhan hiệu dụng
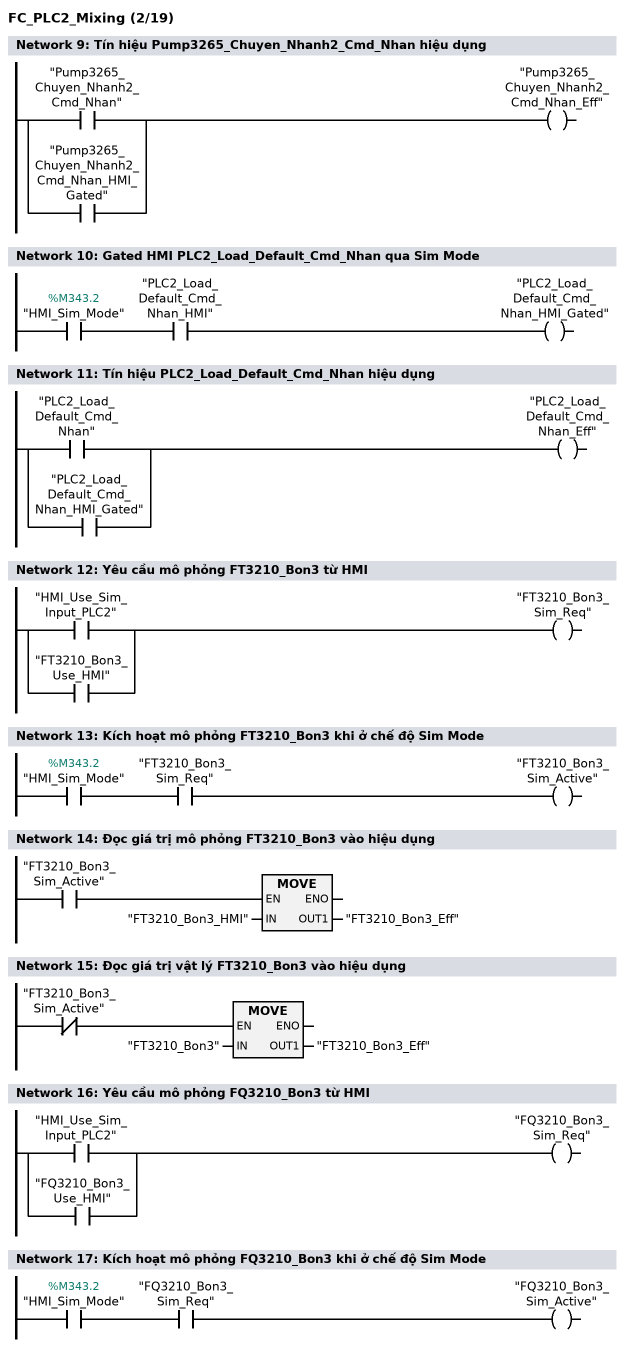
   RUNG wire#powerrail
      Contact( "Pump3265_Chuyen_Nhanh2_Cmd_Nhan" )
      wire#w1
      Coil( "Pump3265_Chuyen_Nhanh2_Cmd_Nhan_Eff" )
   END_RUNG
   RUNG wire#powerrail
      Contact( "Pump3265_Chuyen_Nhanh2_Cmd_Nhan_HMI_Gated" )
   END_RUNG wire#w1
   // the same network as SCL:
   "Pump3265_Chuyen_Nhanh2_Cmd_Nhan_Eff" := "Pump3265_Chuyen_Nhanh2_Cmd_Nhan" OR "Pump3265_Chuyen_Nhanh2_Cmd_Nhan_HMI_Gated";
END_REGION

REGION Network 10: Gated HMI PLC2_Load_Default_Cmd_Nhan qua Sim Mode
   RUNG wire#powerrail
      Contact( "HMI_Sim_Mode" )
      Contact( "PLC2_Load_Default_Cmd_Nhan_HMI" )
      Coil( "PLC2_Load_Default_Cmd_Nhan_HMI_Gated" )
   END_RUNG
   // the same network as SCL:
   "PLC2_Load_Default_Cmd_Nhan_HMI_Gated" := "HMI_Sim_Mode" AND "PLC2_Load_Default_Cmd_Nhan_HMI";
END_REGION

REGION Network 11: Tín hiệu PLC2_Load_Default_Cmd_Nhan hiệu dụng
   RUNG wire#powerrail
      Contact( "PLC2_Load_Default_Cmd_Nhan" )
      wire#w1
      Coil( "PLC2_Load_Default_Cmd_Nhan_Eff" )
   END_RUNG
   RUNG wire#powerrail
      Contact( "PLC2_Load_Default_Cmd_Nhan_HMI_Gated" )
   END_RUNG wire#w1
   // the same network as SCL:
   "PLC2_Load_Default_Cmd_Nhan_Eff" := "PLC2_Load_Default_Cmd_Nhan" OR "PLC2_Load_Default_Cmd_Nhan_HMI_Gated";
END_REGION

REGION Network 12: Yêu cầu mô phỏng FT3210_Bon3 từ HMI
   RUNG wire#powerrail
      Contact( "HMI_Use_Sim_Input_PLC2" )
      wire#w1
      Coil( "FT3210_Bon3_Sim_Req" )
   END_RUNG
   RUNG wire#powerrail
      Contact( "FT3210_Bon3_Use_HMI" )
   END_RUNG wire#w1
   // the same network as SCL:
   "FT3210_Bon3_Sim_Req" := "HMI_Use_Sim_Input_PLC2" OR "FT3210_Bon3_Use_HMI";
END_REGION

REGION Network 13: Kích hoạt mô phỏng FT3210_Bon3 khi ở chế độ Sim Mode
   RUNG wire#powerrail
      Contact( "HMI_Sim_Mode" )
      Contact( "FT3210_Bon3_Sim_Req" )
      Coil( "FT3210_Bon3_Sim_Active" )
   END_RUNG
   // the same network as SCL:
   "FT3210_Bon3_Sim_Active" := "HMI_Sim_Mode" AND "FT3210_Bon3_Sim_Req";
END_REGION

REGION Network 14: Đọc giá trị mô phỏng FT3210_Bon3 vào hiệu dụng
   RUNG wire#powerrail
      Contact( "FT3210_Bon3_Sim_Active" )
      { S7_GenerateENO := "TRUE" } Move(in := "FT3210_Bon3_HMI", out1 => "FT3210_Bon3_Eff")
   END_RUNG
   // the same network as SCL:
   IF "FT3210_Bon3_Sim_Active" THEN "FT3210_Bon3_Eff" := "FT3210_Bon3_HMI"; END_IF;
END_REGION

REGION Network 15: Đọc giá trị vật lý FT3210_Bon3 vào hiệu dụng
   RUNG wire#powerrail
      I_Contact( "FT3210_Bon3_Sim_Active" )
      { S7_GenerateENO := "TRUE" } Move(in := "FT3210_Bon3", out1 => "FT3210_Bon3_Eff")
   END_RUNG
   // the same network as SCL:
   IF NOT "FT3210_Bon3_Sim_Active" THEN "FT3210_Bon3_Eff" := "FT3210_Bon3"; END_IF;
END_REGION

REGION Network 16: Yêu cầu mô phỏng FQ3210_Bon3 từ HMI
   RUNG wire#powerrail
      Contact( "HMI_Use_Sim_Input_PLC2" )
      wire#w1
      Coil( "FQ3210_Bon3_Sim_Req" )
   END_RUNG
   RUNG wire#powerrail
      Contact( "FQ3210_Bon3_Use_HMI" )
   END_RUNG wire#w1
   // the same network as SCL:
   "FQ3210_Bon3_Sim_Req" := "HMI_Use_Sim_Input_PLC2" OR "FQ3210_Bon3_Use_HMI";
END_REGION

REGION Network 17: Kích hoạt mô phỏng FQ3210_Bon3 khi ở chế độ Sim Mode
   RUNG wire#powerrail
      Contact( "HMI_Sim_Mode" )
      Contact( "FQ3210_Bon3_Sim_Req" )
      Coil( "FQ3210_Bon3_Sim_Active" )
   END_RUNG
   // the same network as SCL:
   "FQ3210_Bon3_Sim_Active" := "HMI_Sim_Mode" AND "FQ3210_Bon3_Sim_Req";
END_REGION

REGION Network 18: Đọc giá trị mô phỏng FQ3210_Bon3 vào hiệu dụng
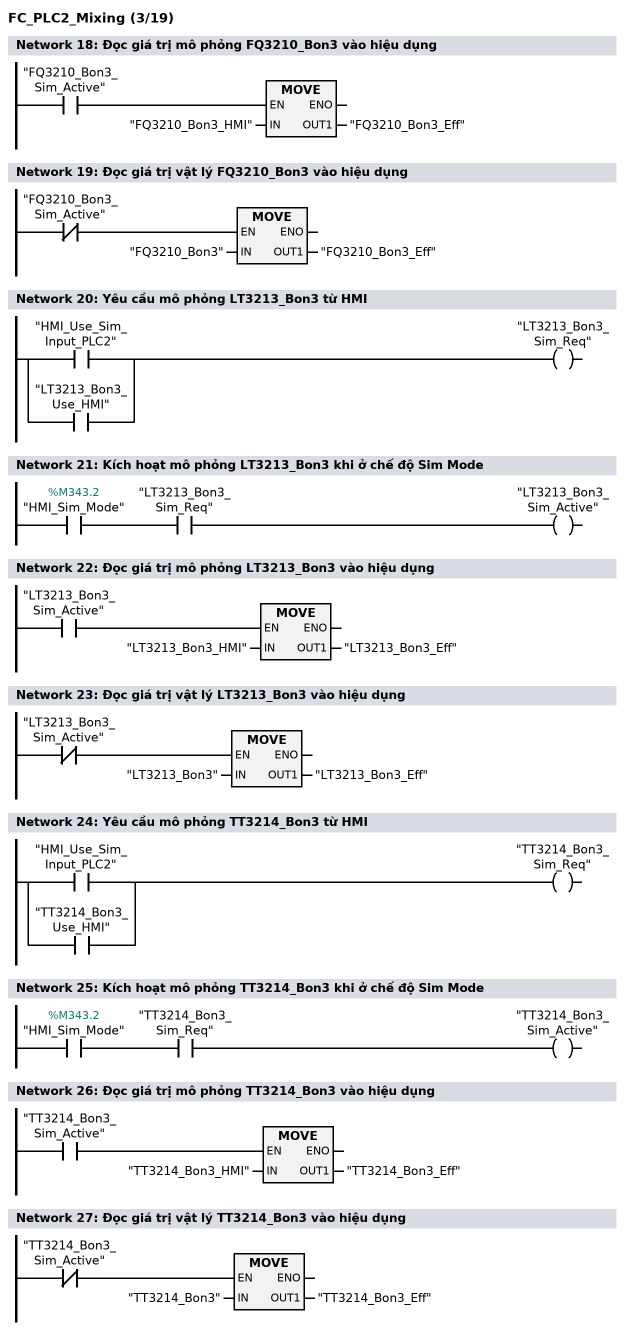
   RUNG wire#powerrail
      Contact( "FQ3210_Bon3_Sim_Active" )
      { S7_GenerateENO := "TRUE" } Move(in := "FQ3210_Bon3_HMI", out1 => "FQ3210_Bon3_Eff")
   END_RUNG
   // the same network as SCL:
   IF "FQ3210_Bon3_Sim_Active" THEN "FQ3210_Bon3_Eff" := "FQ3210_Bon3_HMI"; END_IF;
END_REGION

REGION Network 19: Đọc giá trị vật lý FQ3210_Bon3 vào hiệu dụng
   RUNG wire#powerrail
      I_Contact( "FQ3210_Bon3_Sim_Active" )
      { S7_GenerateENO := "TRUE" } Move(in := "FQ3210_Bon3", out1 => "FQ3210_Bon3_Eff")
   END_RUNG
   // the same network as SCL:
   IF NOT "FQ3210_Bon3_Sim_Active" THEN "FQ3210_Bon3_Eff" := "FQ3210_Bon3"; END_IF;
END_REGION

REGION Network 20: Yêu cầu mô phỏng LT3213_Bon3 từ HMI
   RUNG wire#powerrail
      Contact( "HMI_Use_Sim_Input_PLC2" )
      wire#w1
      Coil( "LT3213_Bon3_Sim_Req" )
   END_RUNG
   RUNG wire#powerrail
      Contact( "LT3213_Bon3_Use_HMI" )
   END_RUNG wire#w1
   // the same network as SCL:
   "LT3213_Bon3_Sim_Req" := "HMI_Use_Sim_Input_PLC2" OR "LT3213_Bon3_Use_HMI";
END_REGION

REGION Network 21: Kích hoạt mô phỏng LT3213_Bon3 khi ở chế độ Sim Mode
   RUNG wire#powerrail
      Contact( "HMI_Sim_Mode" )
      Contact( "LT3213_Bon3_Sim_Req" )
      Coil( "LT3213_Bon3_Sim_Active" )
   END_RUNG
   // the same network as SCL:
   "LT3213_Bon3_Sim_Active" := "HMI_Sim_Mode" AND "LT3213_Bon3_Sim_Req";
END_REGION

REGION Network 22: Đọc giá trị mô phỏng LT3213_Bon3 vào hiệu dụng
   RUNG wire#powerrail
      Contact( "LT3213_Bon3_Sim_Active" )
      { S7_GenerateENO := "TRUE" } Move(in := "LT3213_Bon3_HMI", out1 => "LT3213_Bon3_Eff")
   END_RUNG
   // the same network as SCL:
   IF "LT3213_Bon3_Sim_Active" THEN "LT3213_Bon3_Eff" := "LT3213_Bon3_HMI"; END_IF;
END_REGION

REGION Network 23: Đọc giá trị vật lý LT3213_Bon3 vào hiệu dụng
   RUNG wire#powerrail
      I_Contact( "LT3213_Bon3_Sim_Active" )
      { S7_GenerateENO := "TRUE" } Move(in := "LT3213_Bon3", out1 => "LT3213_Bon3_Eff")
   END_RUNG
   // the same network as SCL:
   IF NOT "LT3213_Bon3_Sim_Active" THEN "LT3213_Bon3_Eff" := "LT3213_Bon3"; END_IF;
END_REGION

REGION Network 24: Yêu cầu mô phỏng TT3214_Bon3 từ HMI
   RUNG wire#powerrail
      Contact( "HMI_Use_Sim_Input_PLC2" )
      wire#w1
      Coil( "TT3214_Bon3_Sim_Req" )
   END_RUNG
   RUNG wire#powerrail
      Contact( "TT3214_Bon3_Use_HMI" )
   END_RUNG wire#w1
   // the same network as SCL:
   "TT3214_Bon3_Sim_Req" := "HMI_Use_Sim_Input_PLC2" OR "TT3214_Bon3_Use_HMI";
END_REGION

REGION Network 25: Kích hoạt mô phỏng TT3214_Bon3 khi ở chế độ Sim Mode
   RUNG wire#powerrail
      Contact( "HMI_Sim_Mode" )
      Contact( "TT3214_Bon3_Sim_Req" )
      Coil( "TT3214_Bon3_Sim_Active" )
   END_RUNG
   // the same network as SCL:
   "TT3214_Bon3_Sim_Active" := "HMI_Sim_Mode" AND "TT3214_Bon3_Sim_Req";
END_REGION

REGION Network 26: Đọc giá trị mô phỏng TT3214_Bon3 vào hiệu dụng
   RUNG wire#powerrail
      Contact( "TT3214_Bon3_Sim_Active" )
      { S7_GenerateENO := "TRUE" } Move(in := "TT3214_Bon3_HMI", out1 => "TT3214_Bon3_Eff")
   END_RUNG
   // the same network as SCL:
   IF "TT3214_Bon3_Sim_Active" THEN "TT3214_Bon3_Eff" := "TT3214_Bon3_HMI"; END_IF;
END_REGION

REGION Network 27: Đọc giá trị vật lý TT3214_Bon3 vào hiệu dụng
   RUNG wire#powerrail
      I_Contact( "TT3214_Bon3_Sim_Active" )
      { S7_GenerateENO := "TRUE" } Move(in := "TT3214_Bon3", out1 => "TT3214_Bon3_Eff")
   END_RUNG
   // the same network as SCL:
   IF NOT "TT3214_Bon3_Sim_Active" THEN "TT3214_Bon3_Eff" := "TT3214_Bon3"; END_IF;
END_REGION

REGION Network 28: Yêu cầu mô phỏng FT3215_Bon4 từ HMI
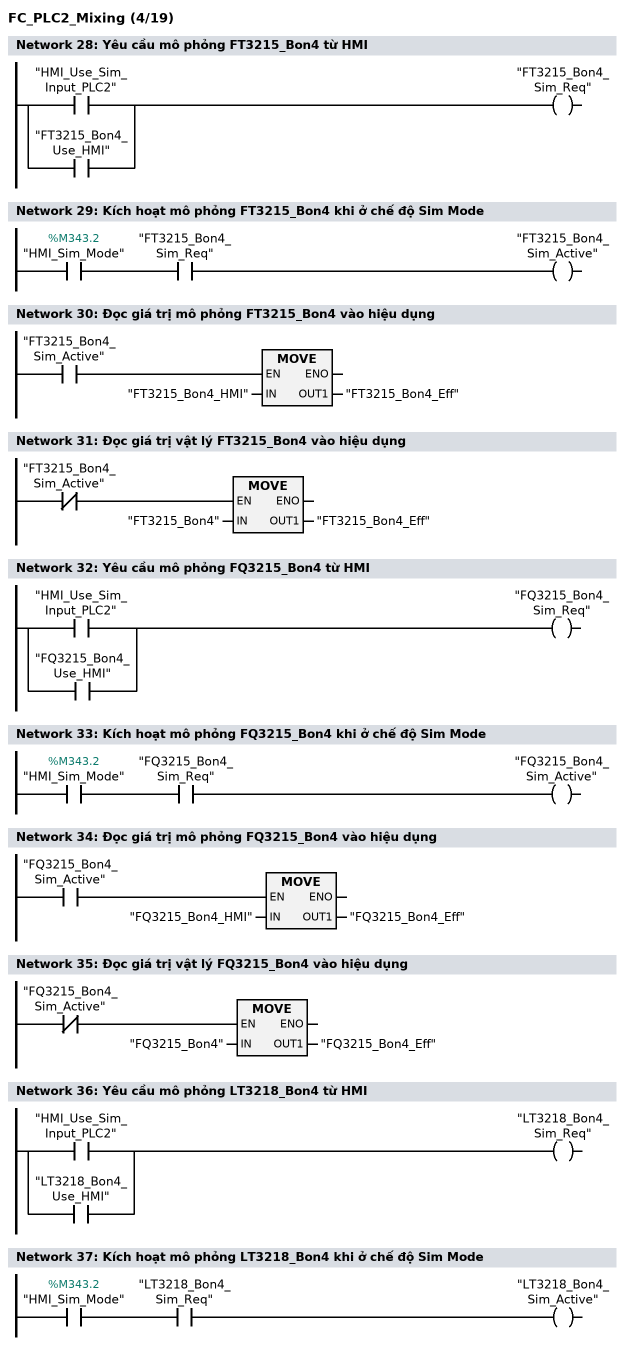
   RUNG wire#powerrail
      Contact( "HMI_Use_Sim_Input_PLC2" )
      wire#w1
      Coil( "FT3215_Bon4_Sim_Req" )
   END_RUNG
   RUNG wire#powerrail
      Contact( "FT3215_Bon4_Use_HMI" )
   END_RUNG wire#w1
   // the same network as SCL:
   "FT3215_Bon4_Sim_Req" := "HMI_Use_Sim_Input_PLC2" OR "FT3215_Bon4_Use_HMI";
END_REGION

REGION Network 29: Kích hoạt mô phỏng FT3215_Bon4 khi ở chế độ Sim Mode
   RUNG wire#powerrail
      Contact( "HMI_Sim_Mode" )
      Contact( "FT3215_Bon4_Sim_Req" )
      Coil( "FT3215_Bon4_Sim_Active" )
   END_RUNG
   // the same network as SCL:
   "FT3215_Bon4_Sim_Active" := "HMI_Sim_Mode" AND "FT3215_Bon4_Sim_Req";
END_REGION

REGION Network 30: Đọc giá trị mô phỏng FT3215_Bon4 vào hiệu dụng
   RUNG wire#powerrail
      Contact( "FT3215_Bon4_Sim_Active" )
      { S7_GenerateENO := "TRUE" } Move(in := "FT3215_Bon4_HMI", out1 => "FT3215_Bon4_Eff")
   END_RUNG
   // the same network as SCL:
   IF "FT3215_Bon4_Sim_Active" THEN "FT3215_Bon4_Eff" := "FT3215_Bon4_HMI"; END_IF;
END_REGION

REGION Network 31: Đọc giá trị vật lý FT3215_Bon4 vào hiệu dụng
   RUNG wire#powerrail
      I_Contact( "FT3215_Bon4_Sim_Active" )
      { S7_GenerateENO := "TRUE" } Move(in := "FT3215_Bon4", out1 => "FT3215_Bon4_Eff")
   END_RUNG
   // the same network as SCL:
   IF NOT "FT3215_Bon4_Sim_Active" THEN "FT3215_Bon4_Eff" := "FT3215_Bon4"; END_IF;
END_REGION

REGION Network 32: Yêu cầu mô phỏng FQ3215_Bon4 từ HMI
   RUNG wire#powerrail
      Contact( "HMI_Use_Sim_Input_PLC2" )
      wire#w1
      Coil( "FQ3215_Bon4_Sim_Req" )
   END_RUNG
   RUNG wire#powerrail
      Contact( "FQ3215_Bon4_Use_HMI" )
   END_RUNG wire#w1
   // the same network as SCL:
   "FQ3215_Bon4_Sim_Req" := "HMI_Use_Sim_Input_PLC2" OR "FQ3215_Bon4_Use_HMI";
END_REGION

REGION Network 33: Kích hoạt mô phỏng FQ3215_Bon4 khi ở chế độ Sim Mode
   RUNG wire#powerrail
      Contact( "HMI_Sim_Mode" )
      Contact( "FQ3215_Bon4_Sim_Req" )
      Coil( "FQ3215_Bon4_Sim_Active" )
   END_RUNG
   // the same network as SCL:
   "FQ3215_Bon4_Sim_Active" := "HMI_Sim_Mode" AND "FQ3215_Bon4_Sim_Req";
END_REGION

REGION Network 34: Đọc giá trị mô phỏng FQ3215_Bon4 vào hiệu dụng
   RUNG wire#powerrail
      Contact( "FQ3215_Bon4_Sim_Active" )
      { S7_GenerateENO := "TRUE" } Move(in := "FQ3215_Bon4_HMI", out1 => "FQ3215_Bon4_Eff")
   END_RUNG
   // the same network as SCL:
   IF "FQ3215_Bon4_Sim_Active" THEN "FQ3215_Bon4_Eff" := "FQ3215_Bon4_HMI"; END_IF;
END_REGION

REGION Network 35: Đọc giá trị vật lý FQ3215_Bon4 vào hiệu dụng
   RUNG wire#powerrail
      I_Contact( "FQ3215_Bon4_Sim_Active" )
      { S7_GenerateENO := "TRUE" } Move(in := "FQ3215_Bon4", out1 => "FQ3215_Bon4_Eff")
   END_RUNG
   // the same network as SCL:
   IF NOT "FQ3215_Bon4_Sim_Active" THEN "FQ3215_Bon4_Eff" := "FQ3215_Bon4"; END_IF;
END_REGION

REGION Network 36: Yêu cầu mô phỏng LT3218_Bon4 từ HMI
   RUNG wire#powerrail
      Contact( "HMI_Use_Sim_Input_PLC2" )
      wire#w1
      Coil( "LT3218_Bon4_Sim_Req" )
   END_RUNG
   RUNG wire#powerrail
      Contact( "LT3218_Bon4_Use_HMI" )
   END_RUNG wire#w1
   // the same network as SCL:
   "LT3218_Bon4_Sim_Req" := "HMI_Use_Sim_Input_PLC2" OR "LT3218_Bon4_Use_HMI";
END_REGION

REGION Network 37: Kích hoạt mô phỏng LT3218_Bon4 khi ở chế độ Sim Mode
   RUNG wire#powerrail
      Contact( "HMI_Sim_Mode" )
      Contact( "LT3218_Bon4_Sim_Req" )
      Coil( "LT3218_Bon4_Sim_Active" )
   END_RUNG
   // the same network as SCL:
   "LT3218_Bon4_Sim_Active" := "HMI_Sim_Mode" AND "LT3218_Bon4_Sim_Req";
END_REGION

REGION Network 38: Đọc giá trị mô phỏng LT3218_Bon4 vào hiệu dụng
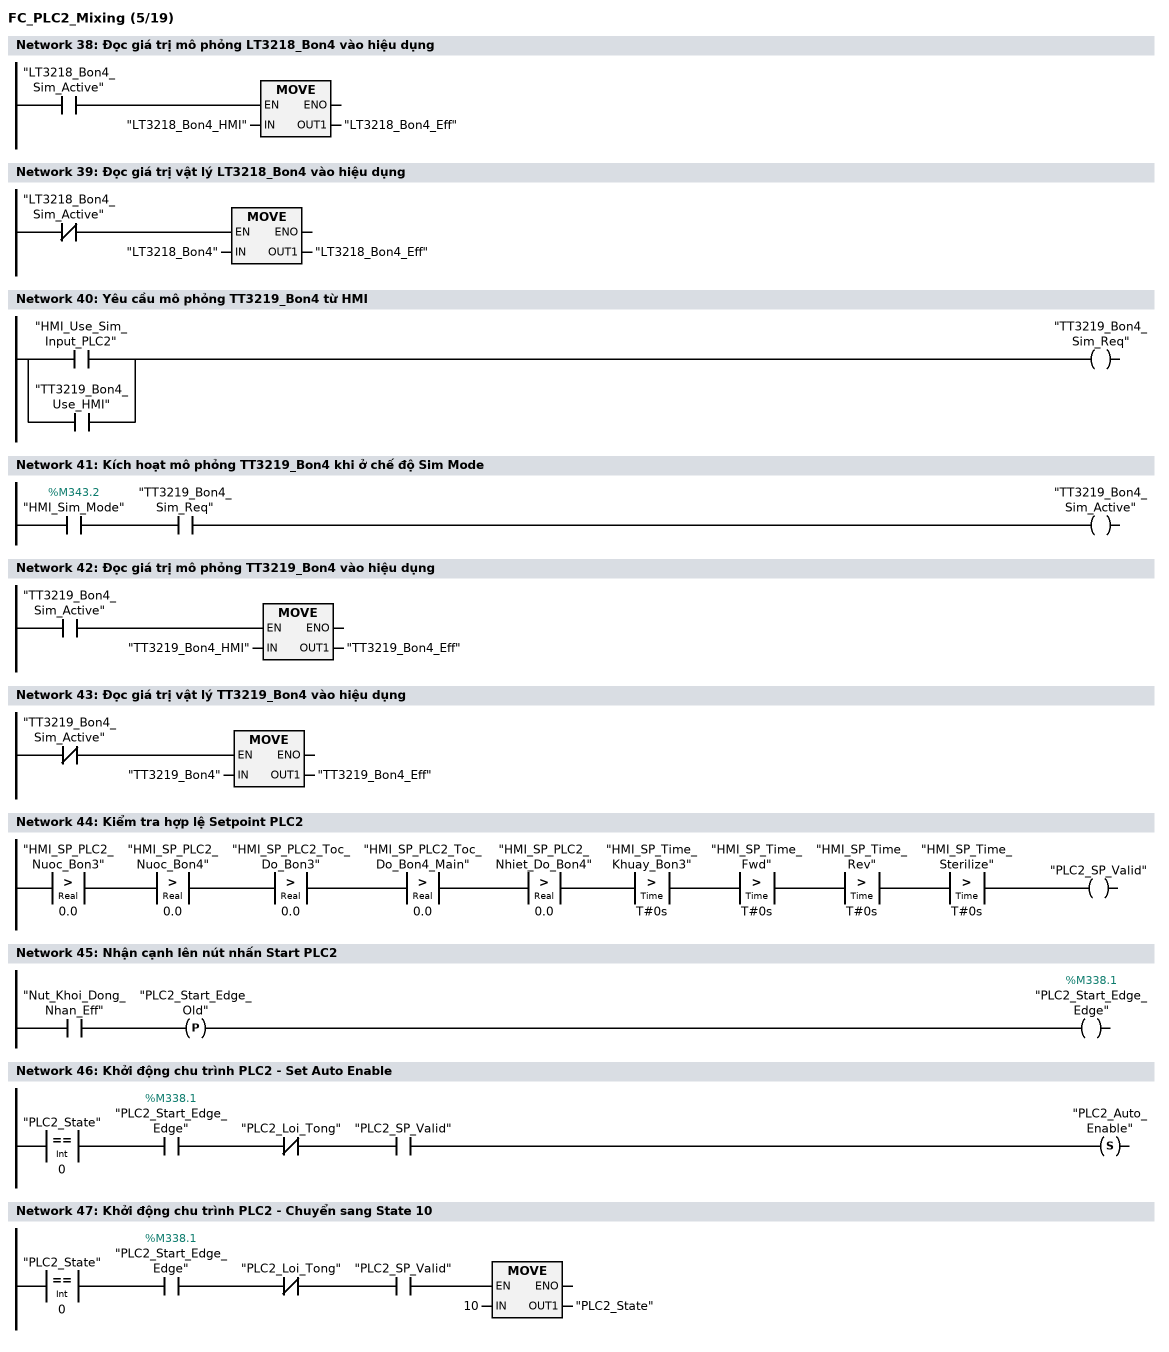
   RUNG wire#powerrail
      Contact( "LT3218_Bon4_Sim_Active" )
      { S7_GenerateENO := "TRUE" } Move(in := "LT3218_Bon4_HMI", out1 => "LT3218_Bon4_Eff")
   END_RUNG
   // the same network as SCL:
   IF "LT3218_Bon4_Sim_Active" THEN "LT3218_Bon4_Eff" := "LT3218_Bon4_HMI"; END_IF;
END_REGION

REGION Network 39: Đọc giá trị vật lý LT3218_Bon4 vào hiệu dụng
   RUNG wire#powerrail
      I_Contact( "LT3218_Bon4_Sim_Active" )
      { S7_GenerateENO := "TRUE" } Move(in := "LT3218_Bon4", out1 => "LT3218_Bon4_Eff")
   END_RUNG
   // the same network as SCL:
   IF NOT "LT3218_Bon4_Sim_Active" THEN "LT3218_Bon4_Eff" := "LT3218_Bon4"; END_IF;
END_REGION

REGION Network 40: Yêu cầu mô phỏng TT3219_Bon4 từ HMI
   RUNG wire#powerrail
      Contact( "HMI_Use_Sim_Input_PLC2" )
      wire#w1
      Coil( "TT3219_Bon4_Sim_Req" )
   END_RUNG
   RUNG wire#powerrail
      Contact( "TT3219_Bon4_Use_HMI" )
   END_RUNG wire#w1
   // the same network as SCL:
   "TT3219_Bon4_Sim_Req" := "HMI_Use_Sim_Input_PLC2" OR "TT3219_Bon4_Use_HMI";
END_REGION

REGION Network 41: Kích hoạt mô phỏng TT3219_Bon4 khi ở chế độ Sim Mode
   RUNG wire#powerrail
      Contact( "HMI_Sim_Mode" )
      Contact( "TT3219_Bon4_Sim_Req" )
      Coil( "TT3219_Bon4_Sim_Active" )
   END_RUNG
   // the same network as SCL:
   "TT3219_Bon4_Sim_Active" := "HMI_Sim_Mode" AND "TT3219_Bon4_Sim_Req";
END_REGION

REGION Network 42: Đọc giá trị mô phỏng TT3219_Bon4 vào hiệu dụng
   RUNG wire#powerrail
      Contact( "TT3219_Bon4_Sim_Active" )
      { S7_GenerateENO := "TRUE" } Move(in := "TT3219_Bon4_HMI", out1 => "TT3219_Bon4_Eff")
   END_RUNG
   // the same network as SCL:
   IF "TT3219_Bon4_Sim_Active" THEN "TT3219_Bon4_Eff" := "TT3219_Bon4_HMI"; END_IF;
END_REGION

REGION Network 43: Đọc giá trị vật lý TT3219_Bon4 vào hiệu dụng
   RUNG wire#powerrail
      I_Contact( "TT3219_Bon4_Sim_Active" )
      { S7_GenerateENO := "TRUE" } Move(in := "TT3219_Bon4", out1 => "TT3219_Bon4_Eff")
   END_RUNG
   // the same network as SCL:
   IF NOT "TT3219_Bon4_Sim_Active" THEN "TT3219_Bon4_Eff" := "TT3219_Bon4"; END_IF;
END_REGION

REGION Network 44: Kiểm tra hợp lệ Setpoint PLC2
   RUNG wire#powerrail
      { S7_Templates := "SrcType := Real" } GT_Contact(in1 := "HMI_SP_PLC2_Nuoc_Bon3", in2 := 0.0)
      { S7_Templates := "SrcType := Real" } GT_Contact(in1 := "HMI_SP_PLC2_Nuoc_Bon4", in2 := 0.0)
      { S7_Templates := "SrcType := Real" } GT_Contact(in1 := "HMI_SP_PLC2_Toc_Do_Bon3", in2 := 0.0)
      { S7_Templates := "SrcType := Real" } GT_Contact(in1 := "HMI_SP_PLC2_Toc_Do_Bon4_Main", in2 := 0.0)
      { S7_Templates := "SrcType := Real" } GT_Contact(in1 := "HMI_SP_PLC2_Nhiet_Do_Bon4", in2 := 0.0)
      { S7_Templates := "SrcType := Time" } GT_Contact(in1 := "HMI_SP_Time_Khuay_Bon3", in2 := T#0s)
      { S7_Templates := "SrcType := Time" } GT_Contact(in1 := "HMI_SP_Time_Fwd", in2 := T#0s)
      { S7_Templates := "SrcType := Time" } GT_Contact(in1 := "HMI_SP_Time_Rev", in2 := T#0s)
      { S7_Templates := "SrcType := Time" } GT_Contact(in1 := "HMI_SP_Time_Sterilize", in2 := T#0s)
      Coil( "PLC2_SP_Valid" )
   END_RUNG
   // the same network as SCL:
   "PLC2_SP_Valid" := ("HMI_SP_PLC2_Nuoc_Bon3" > 0.0) AND ("HMI_SP_PLC2_Nuoc_Bon4" > 0.0) AND ("HMI_SP_PLC2_Toc_Do_Bon3" > 0.0) AND ("HMI_SP_PLC2_Toc_Do_Bon4_Main" > 0.0) AND ("HMI_SP_PLC2_Nhiet_Do_Bon4" > 0.0) AND ("HMI_SP_Time_Khuay_Bon3" > T#0s) AND ("HMI_SP_Time_Fwd" > T#0s) AND ("HMI_SP_Time_Rev" > T#0s) AND ("HMI_SP_Time_Sterilize" > T#0s);
END_REGION

REGION Network 45: Nhận cạnh lên nút nhấn Start PLC2
   RUNG wire#powerrail
      Contact( "Nut_Khoi_Dong_Nhan_Eff" )
      P_Trig( "PLC2_Start_Edge_Old" )
      Coil( "PLC2_Start_Edge_Edge" )
   END_RUNG
   // the same network as SCL:
   #_w1 := "Nut_Khoi_Dong_Nhan_Eff" AND NOT "PLC2_Start_Edge_Old";   // rising edge
   "PLC2_Start_Edge_Old" := "Nut_Khoi_Dong_Nhan_Eff";
   "PLC2_Start_Edge_Edge" := #_w1;
END_REGION

REGION Network 46: Khởi động chu trình PLC2 - Set Auto Enable
   RUNG wire#powerrail
      { S7_Templates := "SrcType := Int" } EQ_Contact(in1 := "PLC2_State", in2 := 0)
      Contact( "PLC2_Start_Edge_Edge" )
      I_Contact( "PLC2_Loi_Tong" )
      Contact( "PLC2_SP_Valid" )
      S_Coil( "PLC2_Auto_Enable" )
   END_RUNG
   // the same network as SCL:
   IF ("PLC2_State" = 0) AND "PLC2_Start_Edge_Edge" AND NOT "PLC2_Loi_Tong" AND "PLC2_SP_Valid" THEN
       "PLC2_Auto_Enable" := TRUE;
   END_IF;
END_REGION

REGION Network 47: Khởi động chu trình PLC2 - Chuyển sang State 10
   RUNG wire#powerrail
      { S7_Templates := "SrcType := Int" } EQ_Contact(in1 := "PLC2_State", in2 := 0)
      Contact( "PLC2_Start_Edge_Edge" )
      I_Contact( "PLC2_Loi_Tong" )
      Contact( "PLC2_SP_Valid" )
      { S7_GenerateENO := "TRUE" } Move(in := 10, out1 => "PLC2_State")
   END_RUNG
   // the same network as SCL:
   IF ("PLC2_State" = 0) AND "PLC2_Start_Edge_Edge" AND NOT "PLC2_Loi_Tong" AND "PLC2_SP_Valid" THEN
       "PLC2_State" := 10;
   END_IF;
END_REGION

REGION Network 48: Báo lỗi setpoint PLC2 khi bấm Start
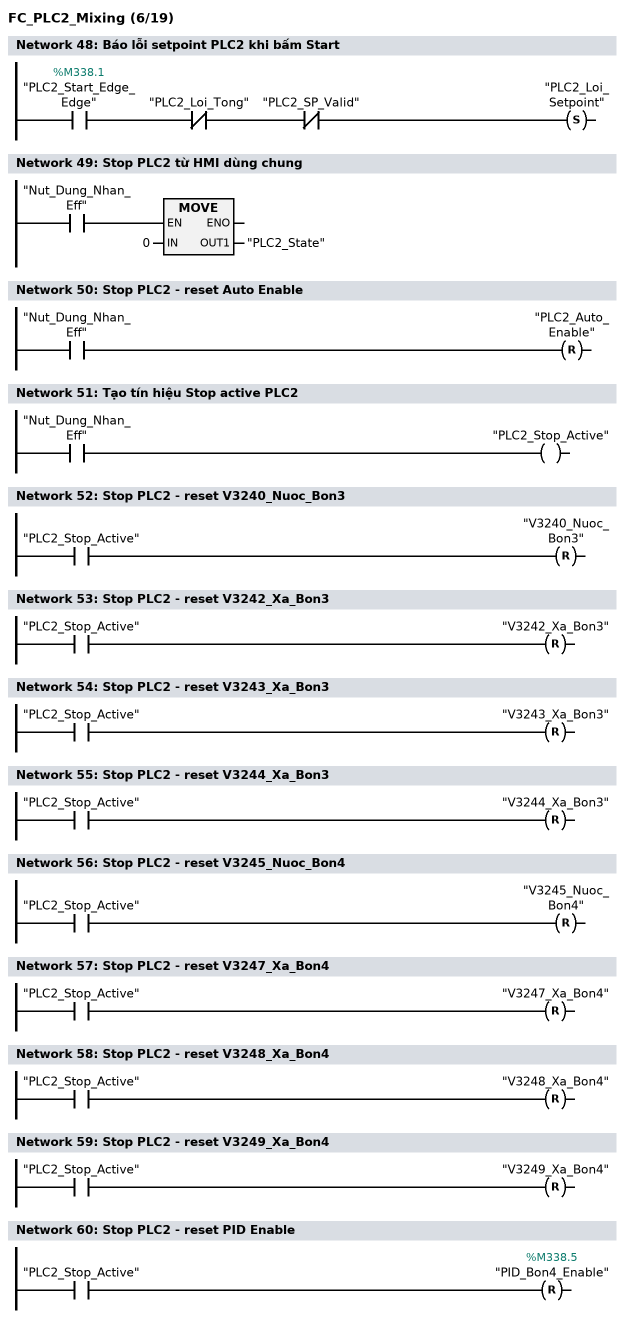
   RUNG wire#powerrail
      Contact( "PLC2_Start_Edge_Edge" )
      I_Contact( "PLC2_Loi_Tong" )
      I_Contact( "PLC2_SP_Valid" )
      S_Coil( "PLC2_Loi_Setpoint" )
   END_RUNG
   // the same network as SCL:
   IF "PLC2_Start_Edge_Edge" AND NOT "PLC2_Loi_Tong" AND NOT "PLC2_SP_Valid" THEN
       "PLC2_Loi_Setpoint" := TRUE;
   END_IF;
END_REGION

REGION Network 49: Stop PLC2 từ HMI dùng chung
   RUNG wire#powerrail
      Contact( "Nut_Dung_Nhan_Eff" )
      { S7_GenerateENO := "TRUE" } Move(in := 0, out1 => "PLC2_State")
   END_RUNG
   // the same network as SCL:
   IF "Nut_Dung_Nhan_Eff" THEN "PLC2_State" := 0; END_IF;
END_REGION

REGION Network 50: Stop PLC2 - reset Auto Enable
   RUNG wire#powerrail
      Contact( "Nut_Dung_Nhan_Eff" )
      R_Coil( "PLC2_Auto_Enable" )
   END_RUNG
   // the same network as SCL:
   IF "Nut_Dung_Nhan_Eff" THEN "PLC2_Auto_Enable" := FALSE; END_IF;
END_REGION

REGION Network 51: Tạo tín hiệu Stop active PLC2
   RUNG wire#powerrail
      Contact( "Nut_Dung_Nhan_Eff" )
      Coil( "PLC2_Stop_Active" )
   END_RUNG
   // the same network as SCL:
   "PLC2_Stop_Active" := "Nut_Dung_Nhan_Eff";
END_REGION

REGION Network 52: Stop PLC2 - reset V3240_Nuoc_Bon3
   RUNG wire#powerrail
      Contact( "PLC2_Stop_Active" )
      R_Coil( "V3240_Nuoc_Bon3" )
   END_RUNG
   // the same network as SCL:
   IF "PLC2_Stop_Active" THEN "V3240_Nuoc_Bon3" := FALSE; END_IF;
END_REGION

REGION Network 53: Stop PLC2 - reset V3242_Xa_Bon3
   RUNG wire#powerrail
      Contact( "PLC2_Stop_Active" )
      R_Coil( "V3242_Xa_Bon3" )
   END_RUNG
   // the same network as SCL:
   IF "PLC2_Stop_Active" THEN "V3242_Xa_Bon3" := FALSE; END_IF;
END_REGION

REGION Network 54: Stop PLC2 - reset V3243_Xa_Bon3
   RUNG wire#powerrail
      Contact( "PLC2_Stop_Active" )
      R_Coil( "V3243_Xa_Bon3" )
   END_RUNG
   // the same network as SCL:
   IF "PLC2_Stop_Active" THEN "V3243_Xa_Bon3" := FALSE; END_IF;
END_REGION

REGION Network 55: Stop PLC2 - reset V3244_Xa_Bon3
   RUNG wire#powerrail
      Contact( "PLC2_Stop_Active" )
      R_Coil( "V3244_Xa_Bon3" )
   END_RUNG
   // the same network as SCL:
   IF "PLC2_Stop_Active" THEN "V3244_Xa_Bon3" := FALSE; END_IF;
END_REGION

REGION Network 56: Stop PLC2 - reset V3245_Nuoc_Bon4
   RUNG wire#powerrail
      Contact( "PLC2_Stop_Active" )
      R_Coil( "V3245_Nuoc_Bon4" )
   END_RUNG
   // the same network as SCL:
   IF "PLC2_Stop_Active" THEN "V3245_Nuoc_Bon4" := FALSE; END_IF;
END_REGION

REGION Network 57: Stop PLC2 - reset V3247_Xa_Bon4
   RUNG wire#powerrail
      Contact( "PLC2_Stop_Active" )
      R_Coil( "V3247_Xa_Bon4" )
   END_RUNG
   // the same network as SCL:
   IF "PLC2_Stop_Active" THEN "V3247_Xa_Bon4" := FALSE; END_IF;
END_REGION

REGION Network 58: Stop PLC2 - reset V3248_Xa_Bon4
   RUNG wire#powerrail
      Contact( "PLC2_Stop_Active" )
      R_Coil( "V3248_Xa_Bon4" )
   END_RUNG
   // the same network as SCL:
   IF "PLC2_Stop_Active" THEN "V3248_Xa_Bon4" := FALSE; END_IF;
END_REGION

REGION Network 59: Stop PLC2 - reset V3249_Xa_Bon4
   RUNG wire#powerrail
      Contact( "PLC2_Stop_Active" )
      R_Coil( "V3249_Xa_Bon4" )
   END_RUNG
   // the same network as SCL:
   IF "PLC2_Stop_Active" THEN "V3249_Xa_Bon4" := FALSE; END_IF;
END_REGION

REGION Network 60: Stop PLC2 - reset PID Enable
   RUNG wire#powerrail
      Contact( "PLC2_Stop_Active" )
      R_Coil( "PID_Bon4_Enable" )
   END_RUNG
   // the same network as SCL:
   IF "PLC2_Stop_Active" THEN "PID_Bon4_Enable" := FALSE; END_IF;
END_REGION

REGION Network 61: Stop PLC2 - clear CV3211_Nuoc_Bon3
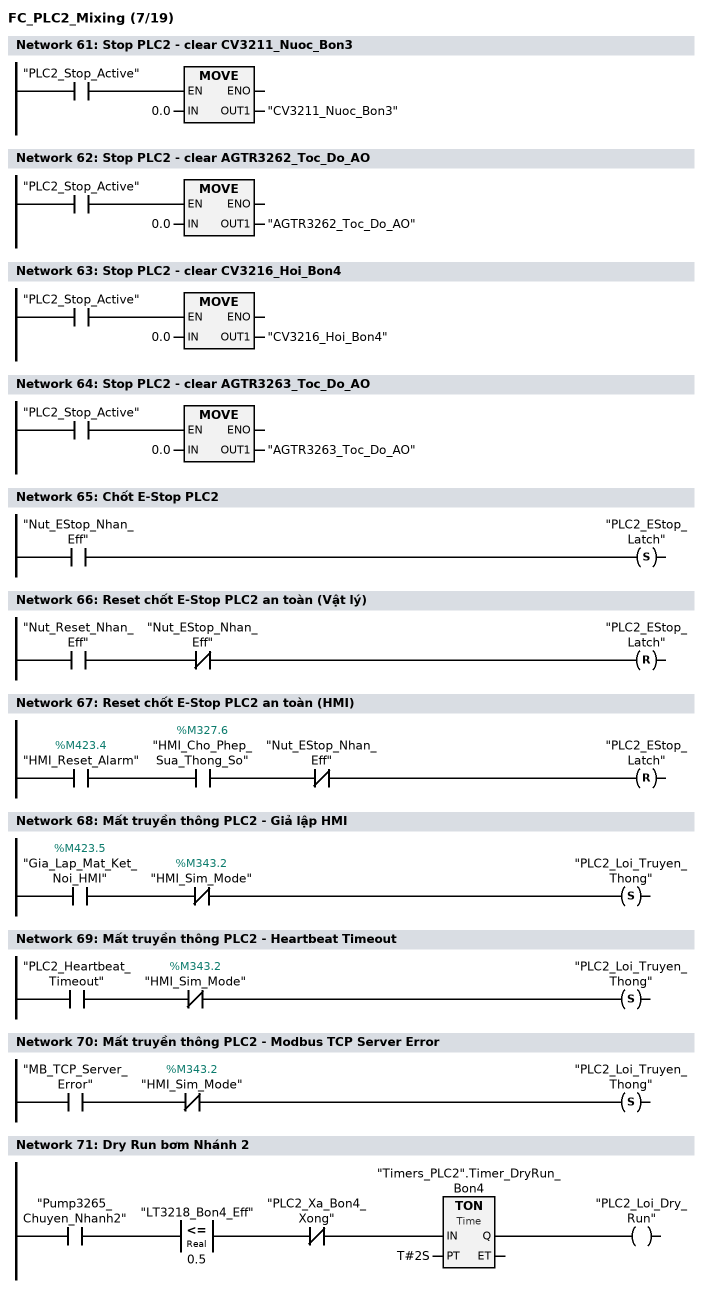
   RUNG wire#powerrail
      Contact( "PLC2_Stop_Active" )
      { S7_GenerateENO := "TRUE" } Move(in := 0.0, out1 => "CV3211_Nuoc_Bon3")
   END_RUNG
   // the same network as SCL:
   IF "PLC2_Stop_Active" THEN "CV3211_Nuoc_Bon3" := 0.0; END_IF;
END_REGION

REGION Network 62: Stop PLC2 - clear AGTR3262_Toc_Do_AO
   RUNG wire#powerrail
      Contact( "PLC2_Stop_Active" )
      { S7_GenerateENO := "TRUE" } Move(in := 0.0, out1 => "AGTR3262_Toc_Do_AO")
   END_RUNG
   // the same network as SCL:
   IF "PLC2_Stop_Active" THEN "AGTR3262_Toc_Do_AO" := 0.0; END_IF;
END_REGION

REGION Network 63: Stop PLC2 - clear CV3216_Hoi_Bon4
   RUNG wire#powerrail
      Contact( "PLC2_Stop_Active" )
      { S7_GenerateENO := "TRUE" } Move(in := 0.0, out1 => "CV3216_Hoi_Bon4")
   END_RUNG
   // the same network as SCL:
   IF "PLC2_Stop_Active" THEN "CV3216_Hoi_Bon4" := 0.0; END_IF;
END_REGION

REGION Network 64: Stop PLC2 - clear AGTR3263_Toc_Do_AO
   RUNG wire#powerrail
      Contact( "PLC2_Stop_Active" )
      { S7_GenerateENO := "TRUE" } Move(in := 0.0, out1 => "AGTR3263_Toc_Do_AO")
   END_RUNG
   // the same network as SCL:
   IF "PLC2_Stop_Active" THEN "AGTR3263_Toc_Do_AO" := 0.0; END_IF;
END_REGION

REGION Network 65: Chốt E-Stop PLC2
   RUNG wire#powerrail
      Contact( "Nut_EStop_Nhan_Eff" )
      S_Coil( "PLC2_EStop_Latch" )
   END_RUNG
   // the same network as SCL:
   IF "Nut_EStop_Nhan_Eff" THEN "PLC2_EStop_Latch" := TRUE; END_IF;
END_REGION

REGION Network 66: Reset chốt E-Stop PLC2 an toàn (Vật lý)
   RUNG wire#powerrail
      Contact( "Nut_Reset_Nhan_Eff" )
      I_Contact( "Nut_EStop_Nhan_Eff" )
      R_Coil( "PLC2_EStop_Latch" )
   END_RUNG
   // the same network as SCL:
   IF "Nut_Reset_Nhan_Eff" AND NOT "Nut_EStop_Nhan_Eff" THEN "PLC2_EStop_Latch" := FALSE; END_IF;
END_REGION

REGION Network 67: Reset chốt E-Stop PLC2 an toàn (HMI)
   RUNG wire#powerrail
      Contact( "HMI_Reset_Alarm" )
      Contact( "HMI_Cho_Phep_Sua_Thong_So" )
      I_Contact( "Nut_EStop_Nhan_Eff" )
      R_Coil( "PLC2_EStop_Latch" )
   END_RUNG
   // the same network as SCL:
   IF "HMI_Reset_Alarm" AND "HMI_Cho_Phep_Sua_Thong_So" AND NOT "Nut_EStop_Nhan_Eff" THEN
       "PLC2_EStop_Latch" := FALSE;
   END_IF;
END_REGION

REGION Network 68: Mất truyền thông PLC2 - Giả lập HMI
   RUNG wire#powerrail
      Contact( "Gia_Lap_Mat_Ket_Noi_HMI" )
      I_Contact( "HMI_Sim_Mode" )
      S_Coil( "PLC2_Loi_Truyen_Thong" )
   END_RUNG
   // the same network as SCL:
   IF "Gia_Lap_Mat_Ket_Noi_HMI" AND NOT "HMI_Sim_Mode" THEN "PLC2_Loi_Truyen_Thong" := TRUE; END_IF;
END_REGION

REGION Network 69: Mất truyền thông PLC2 - Heartbeat Timeout
   RUNG wire#powerrail
      Contact( "PLC2_Heartbeat_Timeout" )
      I_Contact( "HMI_Sim_Mode" )
      S_Coil( "PLC2_Loi_Truyen_Thong" )
   END_RUNG
   // the same network as SCL:
   IF "PLC2_Heartbeat_Timeout" AND NOT "HMI_Sim_Mode" THEN "PLC2_Loi_Truyen_Thong" := TRUE; END_IF;
END_REGION

REGION Network 70: Mất truyền thông PLC2 - Modbus TCP Server Error
   RUNG wire#powerrail
      Contact( "MB_TCP_Server_Error" )
      I_Contact( "HMI_Sim_Mode" )
      S_Coil( "PLC2_Loi_Truyen_Thong" )
   END_RUNG
   // the same network as SCL:
   IF "MB_TCP_Server_Error" AND NOT "HMI_Sim_Mode" THEN "PLC2_Loi_Truyen_Thong" := TRUE; END_IF;
END_REGION

REGION Network 71: Dry Run bơm Nhánh 2
   RUNG wire#powerrail
      Contact( "Pump3265_Chuyen_Nhanh2" )
      { S7_Templates := "SrcType := Real" } LE_Contact(in1 := "LT3218_Bon4_Eff", in2 := 0.5)
      I_Contact( "PLC2_Xa_Bon4_Xong" )
      { S7_Templates := "time_type := Time" } "Timers_PLC2".Timer_DryRun_Bon4.TON(pt := T#2S, et =>)
      Coil( "PLC2_Loi_Dry_Run" )
   END_RUNG
   // the same network as SCL:
   "Timers_PLC2".Timer_DryRun_Bon4.TON(IN := "Pump3265_Chuyen_Nhanh2" AND ("LT3218_Bon4_Eff" <= 0.5) AND NOT "PLC2_Xa_Bon4_Xong",
                           PT := T#2S);
   "PLC2_Loi_Dry_Run" := "Timers_PLC2".Timer_DryRun_Bon4.Q;
END_REGION

REGION Network 72: Dosing Bồn 3 lỗi quá 5 giây không có lưu lượng
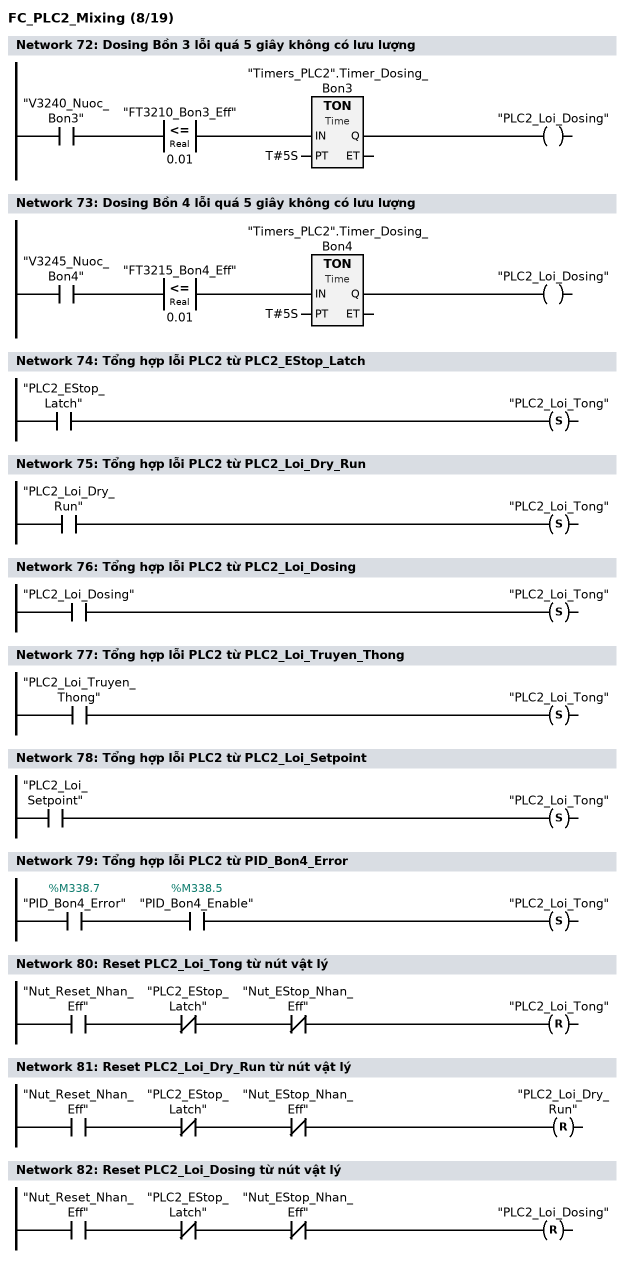
   RUNG wire#powerrail
      Contact( "V3240_Nuoc_Bon3" )
      { S7_Templates := "SrcType := Real" } LE_Contact(in1 := "FT3210_Bon3_Eff", in2 := 0.01)
      { S7_Templates := "time_type := Time" } "Timers_PLC2".Timer_Dosing_Bon3.TON(pt := T#5S, et =>)
      Coil( "PLC2_Loi_Dosing" )
   END_RUNG
   // the same network as SCL:
   "Timers_PLC2".Timer_Dosing_Bon3.TON(IN := "V3240_Nuoc_Bon3" AND ("FT3210_Bon3_Eff" <= 0.01), PT := T#5S);
   "PLC2_Loi_Dosing" := "Timers_PLC2".Timer_Dosing_Bon3.Q;
END_REGION

REGION Network 73: Dosing Bồn 4 lỗi quá 5 giây không có lưu lượng
   RUNG wire#powerrail
      Contact( "V3245_Nuoc_Bon4" )
      { S7_Templates := "SrcType := Real" } LE_Contact(in1 := "FT3215_Bon4_Eff", in2 := 0.01)
      { S7_Templates := "time_type := Time" } "Timers_PLC2".Timer_Dosing_Bon4.TON(pt := T#5S, et =>)
      Coil( "PLC2_Loi_Dosing" )
   END_RUNG
   // the same network as SCL:
   "Timers_PLC2".Timer_Dosing_Bon4.TON(IN := "V3245_Nuoc_Bon4" AND ("FT3215_Bon4_Eff" <= 0.01), PT := T#5S);
   "PLC2_Loi_Dosing" := "Timers_PLC2".Timer_Dosing_Bon4.Q;
END_REGION

REGION Network 74: Tổng hợp lỗi PLC2 từ PLC2_EStop_Latch
   RUNG wire#powerrail
      Contact( "PLC2_EStop_Latch" )
      S_Coil( "PLC2_Loi_Tong" )
   END_RUNG
   // the same network as SCL:
   IF "PLC2_EStop_Latch" THEN "PLC2_Loi_Tong" := TRUE; END_IF;
END_REGION

REGION Network 75: Tổng hợp lỗi PLC2 từ PLC2_Loi_Dry_Run
   RUNG wire#powerrail
      Contact( "PLC2_Loi_Dry_Run" )
      S_Coil( "PLC2_Loi_Tong" )
   END_RUNG
   // the same network as SCL:
   IF "PLC2_Loi_Dry_Run" THEN "PLC2_Loi_Tong" := TRUE; END_IF;
END_REGION

REGION Network 76: Tổng hợp lỗi PLC2 từ PLC2_Loi_Dosing
   RUNG wire#powerrail
      Contact( "PLC2_Loi_Dosing" )
      S_Coil( "PLC2_Loi_Tong" )
   END_RUNG
   // the same network as SCL:
   IF "PLC2_Loi_Dosing" THEN "PLC2_Loi_Tong" := TRUE; END_IF;
END_REGION

REGION Network 77: Tổng hợp lỗi PLC2 từ PLC2_Loi_Truyen_Thong
   RUNG wire#powerrail
      Contact( "PLC2_Loi_Truyen_Thong" )
      S_Coil( "PLC2_Loi_Tong" )
   END_RUNG
   // the same network as SCL:
   IF "PLC2_Loi_Truyen_Thong" THEN "PLC2_Loi_Tong" := TRUE; END_IF;
END_REGION

REGION Network 78: Tổng hợp lỗi PLC2 từ PLC2_Loi_Setpoint
   RUNG wire#powerrail
      Contact( "PLC2_Loi_Setpoint" )
      S_Coil( "PLC2_Loi_Tong" )
   END_RUNG
   // the same network as SCL:
   IF "PLC2_Loi_Setpoint" THEN "PLC2_Loi_Tong" := TRUE; END_IF;
END_REGION

REGION Network 79: Tổng hợp lỗi PLC2 từ PID_Bon4_Error
   RUNG wire#powerrail
      Contact( "PID_Bon4_Error" )
      Contact( "PID_Bon4_Enable" )
      S_Coil( "PLC2_Loi_Tong" )
   END_RUNG
   // the same network as SCL:
   IF "PID_Bon4_Error" AND "PID_Bon4_Enable" THEN "PLC2_Loi_Tong" := TRUE; END_IF;
END_REGION

REGION Network 80: Reset PLC2_Loi_Tong từ nút vật lý
   RUNG wire#powerrail
      Contact( "Nut_Reset_Nhan_Eff" )
      I_Contact( "PLC2_EStop_Latch" )
      I_Contact( "Nut_EStop_Nhan_Eff" )
      R_Coil( "PLC2_Loi_Tong" )
   END_RUNG
   // the same network as SCL:
   IF "Nut_Reset_Nhan_Eff" AND NOT "PLC2_EStop_Latch" AND NOT "Nut_EStop_Nhan_Eff" THEN
       "PLC2_Loi_Tong" := FALSE;
   END_IF;
END_REGION

REGION Network 81: Reset PLC2_Loi_Dry_Run từ nút vật lý
   RUNG wire#powerrail
      Contact( "Nut_Reset_Nhan_Eff" )
      I_Contact( "PLC2_EStop_Latch" )
      I_Contact( "Nut_EStop_Nhan_Eff" )
      R_Coil( "PLC2_Loi_Dry_Run" )
   END_RUNG
   // the same network as SCL:
   IF "Nut_Reset_Nhan_Eff" AND NOT "PLC2_EStop_Latch" AND NOT "Nut_EStop_Nhan_Eff" THEN
       "PLC2_Loi_Dry_Run" := FALSE;
   END_IF;
END_REGION

REGION Network 82: Reset PLC2_Loi_Dosing từ nút vật lý
   RUNG wire#powerrail
      Contact( "Nut_Reset_Nhan_Eff" )
      I_Contact( "PLC2_EStop_Latch" )
      I_Contact( "Nut_EStop_Nhan_Eff" )
      R_Coil( "PLC2_Loi_Dosing" )
   END_RUNG
   // the same network as SCL:
   IF "Nut_Reset_Nhan_Eff" AND NOT "PLC2_EStop_Latch" AND NOT "Nut_EStop_Nhan_Eff" THEN
       "PLC2_Loi_Dosing" := FALSE;
   END_IF;
END_REGION

REGION Network 83: Reset PLC2_Loi_Truyen_Thong từ nút vật lý
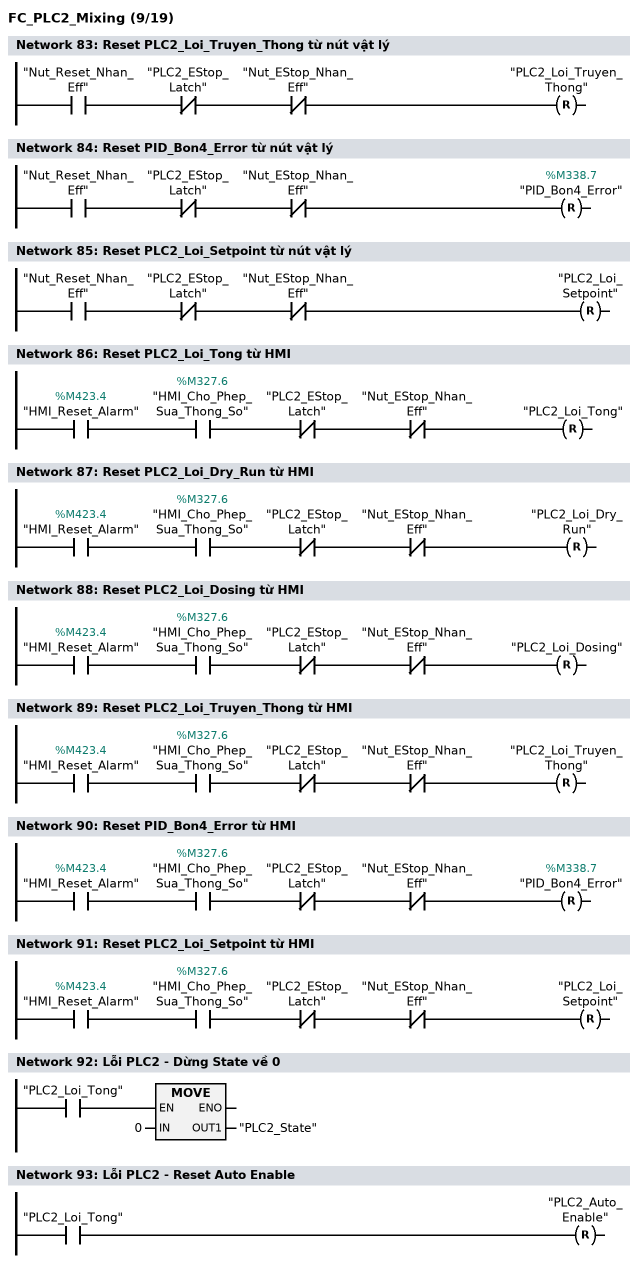
   RUNG wire#powerrail
      Contact( "Nut_Reset_Nhan_Eff" )
      I_Contact( "PLC2_EStop_Latch" )
      I_Contact( "Nut_EStop_Nhan_Eff" )
      R_Coil( "PLC2_Loi_Truyen_Thong" )
   END_RUNG
   // the same network as SCL:
   IF "Nut_Reset_Nhan_Eff" AND NOT "PLC2_EStop_Latch" AND NOT "Nut_EStop_Nhan_Eff" THEN
       "PLC2_Loi_Truyen_Thong" := FALSE;
   END_IF;
END_REGION

REGION Network 84: Reset PID_Bon4_Error từ nút vật lý
   RUNG wire#powerrail
      Contact( "Nut_Reset_Nhan_Eff" )
      I_Contact( "PLC2_EStop_Latch" )
      I_Contact( "Nut_EStop_Nhan_Eff" )
      R_Coil( "PID_Bon4_Error" )
   END_RUNG
   // the same network as SCL:
   IF "Nut_Reset_Nhan_Eff" AND NOT "PLC2_EStop_Latch" AND NOT "Nut_EStop_Nhan_Eff" THEN
       "PID_Bon4_Error" := FALSE;
   END_IF;
END_REGION

REGION Network 85: Reset PLC2_Loi_Setpoint từ nút vật lý
   RUNG wire#powerrail
      Contact( "Nut_Reset_Nhan_Eff" )
      I_Contact( "PLC2_EStop_Latch" )
      I_Contact( "Nut_EStop_Nhan_Eff" )
      R_Coil( "PLC2_Loi_Setpoint" )
   END_RUNG
   // the same network as SCL:
   IF "Nut_Reset_Nhan_Eff" AND NOT "PLC2_EStop_Latch" AND NOT "Nut_EStop_Nhan_Eff" THEN
       "PLC2_Loi_Setpoint" := FALSE;
   END_IF;
END_REGION

REGION Network 86: Reset PLC2_Loi_Tong từ HMI
   RUNG wire#powerrail
      Contact( "HMI_Reset_Alarm" )
      Contact( "HMI_Cho_Phep_Sua_Thong_So" )
      I_Contact( "PLC2_EStop_Latch" )
      I_Contact( "Nut_EStop_Nhan_Eff" )
      R_Coil( "PLC2_Loi_Tong" )
   END_RUNG
   // the same network as SCL:
   IF "HMI_Reset_Alarm" AND "HMI_Cho_Phep_Sua_Thong_So" AND NOT "PLC2_EStop_Latch" AND NOT "Nut_EStop_Nhan_Eff" THEN
       "PLC2_Loi_Tong" := FALSE;
   END_IF;
END_REGION

REGION Network 87: Reset PLC2_Loi_Dry_Run từ HMI
   RUNG wire#powerrail
      Contact( "HMI_Reset_Alarm" )
      Contact( "HMI_Cho_Phep_Sua_Thong_So" )
      I_Contact( "PLC2_EStop_Latch" )
      I_Contact( "Nut_EStop_Nhan_Eff" )
      R_Coil( "PLC2_Loi_Dry_Run" )
   END_RUNG
   // the same network as SCL:
   IF "HMI_Reset_Alarm" AND "HMI_Cho_Phep_Sua_Thong_So" AND NOT "PLC2_EStop_Latch" AND NOT "Nut_EStop_Nhan_Eff" THEN
       "PLC2_Loi_Dry_Run" := FALSE;
   END_IF;
END_REGION

REGION Network 88: Reset PLC2_Loi_Dosing từ HMI
   RUNG wire#powerrail
      Contact( "HMI_Reset_Alarm" )
      Contact( "HMI_Cho_Phep_Sua_Thong_So" )
      I_Contact( "PLC2_EStop_Latch" )
      I_Contact( "Nut_EStop_Nhan_Eff" )
      R_Coil( "PLC2_Loi_Dosing" )
   END_RUNG
   // the same network as SCL:
   IF "HMI_Reset_Alarm" AND "HMI_Cho_Phep_Sua_Thong_So" AND NOT "PLC2_EStop_Latch" AND NOT "Nut_EStop_Nhan_Eff" THEN
       "PLC2_Loi_Dosing" := FALSE;
   END_IF;
END_REGION

REGION Network 89: Reset PLC2_Loi_Truyen_Thong từ HMI
   RUNG wire#powerrail
      Contact( "HMI_Reset_Alarm" )
      Contact( "HMI_Cho_Phep_Sua_Thong_So" )
      I_Contact( "PLC2_EStop_Latch" )
      I_Contact( "Nut_EStop_Nhan_Eff" )
      R_Coil( "PLC2_Loi_Truyen_Thong" )
   END_RUNG
   // the same network as SCL:
   IF "HMI_Reset_Alarm" AND "HMI_Cho_Phep_Sua_Thong_So" AND NOT "PLC2_EStop_Latch" AND NOT "Nut_EStop_Nhan_Eff" THEN
       "PLC2_Loi_Truyen_Thong" := FALSE;
   END_IF;
END_REGION

REGION Network 90: Reset PID_Bon4_Error từ HMI
   RUNG wire#powerrail
      Contact( "HMI_Reset_Alarm" )
      Contact( "HMI_Cho_Phep_Sua_Thong_So" )
      I_Contact( "PLC2_EStop_Latch" )
      I_Contact( "Nut_EStop_Nhan_Eff" )
      R_Coil( "PID_Bon4_Error" )
   END_RUNG
   // the same network as SCL:
   IF "HMI_Reset_Alarm" AND "HMI_Cho_Phep_Sua_Thong_So" AND NOT "PLC2_EStop_Latch" AND NOT "Nut_EStop_Nhan_Eff" THEN
       "PID_Bon4_Error" := FALSE;
   END_IF;
END_REGION

REGION Network 91: Reset PLC2_Loi_Setpoint từ HMI
   RUNG wire#powerrail
      Contact( "HMI_Reset_Alarm" )
      Contact( "HMI_Cho_Phep_Sua_Thong_So" )
      I_Contact( "PLC2_EStop_Latch" )
      I_Contact( "Nut_EStop_Nhan_Eff" )
      R_Coil( "PLC2_Loi_Setpoint" )
   END_RUNG
   // the same network as SCL:
   IF "HMI_Reset_Alarm" AND "HMI_Cho_Phep_Sua_Thong_So" AND NOT "PLC2_EStop_Latch" AND NOT "Nut_EStop_Nhan_Eff" THEN
       "PLC2_Loi_Setpoint" := FALSE;
   END_IF;
END_REGION

REGION Network 92: Lỗi PLC2 - Dừng State về 0
   RUNG wire#powerrail
      Contact( "PLC2_Loi_Tong" )
      { S7_GenerateENO := "TRUE" } Move(in := 0, out1 => "PLC2_State")
   END_RUNG
   // the same network as SCL:
   IF "PLC2_Loi_Tong" THEN "PLC2_State" := 0; END_IF;
END_REGION

REGION Network 93: Lỗi PLC2 - Reset Auto Enable
   RUNG wire#powerrail
      Contact( "PLC2_Loi_Tong" )
      R_Coil( "PLC2_Auto_Enable" )
   END_RUNG
   // the same network as SCL:
   IF "PLC2_Loi_Tong" THEN "PLC2_Auto_Enable" := FALSE; END_IF;
END_REGION

REGION Network 94: Lỗi PLC2 - Reset PID Enable
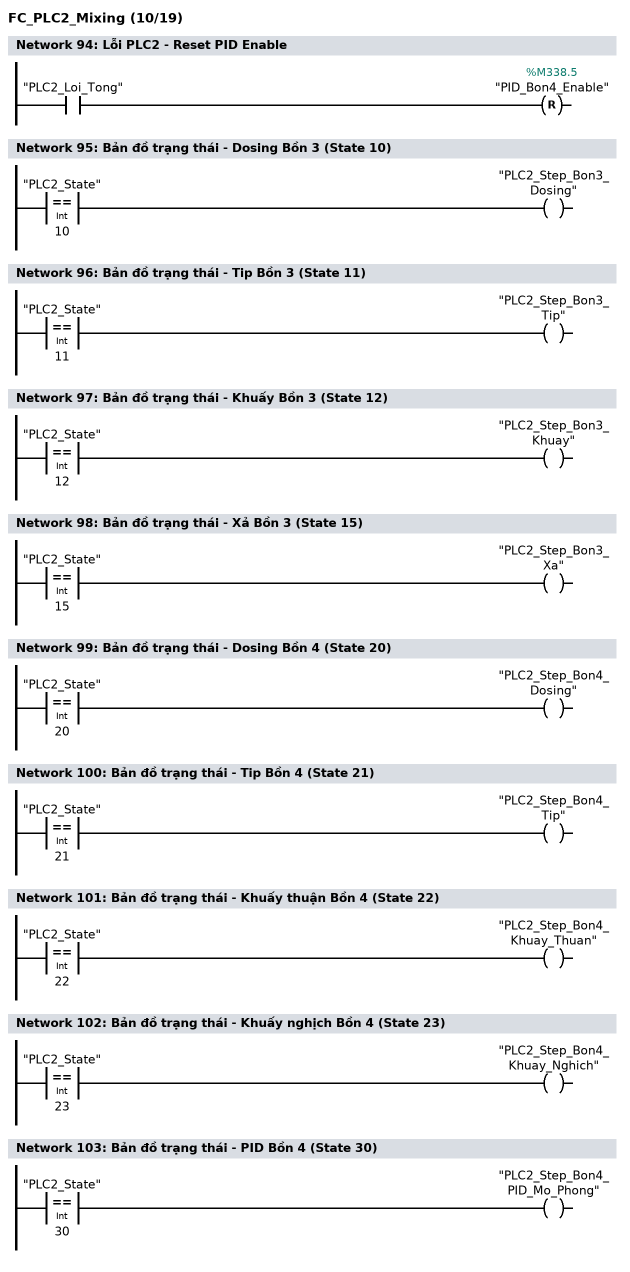
   RUNG wire#powerrail
      Contact( "PLC2_Loi_Tong" )
      R_Coil( "PID_Bon4_Enable" )
   END_RUNG
   // the same network as SCL:
   IF "PLC2_Loi_Tong" THEN "PID_Bon4_Enable" := FALSE; END_IF;
END_REGION

REGION Network 95: Bản đồ trạng thái - Dosing Bồn 3 (State 10)
   RUNG wire#powerrail
      { S7_Templates := "SrcType := Int" } EQ_Contact(in1 := "PLC2_State", in2 := 10)
      Coil( "PLC2_Step_Bon3_Dosing" )
   END_RUNG
   // the same network as SCL:
   "PLC2_Step_Bon3_Dosing" := "PLC2_State" = 10;
END_REGION

REGION Network 96: Bản đồ trạng thái - Tip Bồn 3 (State 11)
   RUNG wire#powerrail
      { S7_Templates := "SrcType := Int" } EQ_Contact(in1 := "PLC2_State", in2 := 11)
      Coil( "PLC2_Step_Bon3_Tip" )
   END_RUNG
   // the same network as SCL:
   "PLC2_Step_Bon3_Tip" := "PLC2_State" = 11;
END_REGION

REGION Network 97: Bản đồ trạng thái - Khuấy Bồn 3 (State 12)
   RUNG wire#powerrail
      { S7_Templates := "SrcType := Int" } EQ_Contact(in1 := "PLC2_State", in2 := 12)
      Coil( "PLC2_Step_Bon3_Khuay" )
   END_RUNG
   // the same network as SCL:
   "PLC2_Step_Bon3_Khuay" := "PLC2_State" = 12;
END_REGION

REGION Network 98: Bản đồ trạng thái - Xả Bồn 3 (State 15)
   RUNG wire#powerrail
      { S7_Templates := "SrcType := Int" } EQ_Contact(in1 := "PLC2_State", in2 := 15)
      Coil( "PLC2_Step_Bon3_Xa" )
   END_RUNG
   // the same network as SCL:
   "PLC2_Step_Bon3_Xa" := "PLC2_State" = 15;
END_REGION

REGION Network 99: Bản đồ trạng thái - Dosing Bồn 4 (State 20)
   RUNG wire#powerrail
      { S7_Templates := "SrcType := Int" } EQ_Contact(in1 := "PLC2_State", in2 := 20)
      Coil( "PLC2_Step_Bon4_Dosing" )
   END_RUNG
   // the same network as SCL:
   "PLC2_Step_Bon4_Dosing" := "PLC2_State" = 20;
END_REGION

REGION Network 100: Bản đồ trạng thái - Tip Bồn 4 (State 21)
   RUNG wire#powerrail
      { S7_Templates := "SrcType := Int" } EQ_Contact(in1 := "PLC2_State", in2 := 21)
      Coil( "PLC2_Step_Bon4_Tip" )
   END_RUNG
   // the same network as SCL:
   "PLC2_Step_Bon4_Tip" := "PLC2_State" = 21;
END_REGION

REGION Network 101: Bản đồ trạng thái - Khuấy thuận Bồn 4 (State 22)
   RUNG wire#powerrail
      { S7_Templates := "SrcType := Int" } EQ_Contact(in1 := "PLC2_State", in2 := 22)
      Coil( "PLC2_Step_Bon4_Khuay_Thuan" )
   END_RUNG
   // the same network as SCL:
   "PLC2_Step_Bon4_Khuay_Thuan" := "PLC2_State" = 22;
END_REGION

REGION Network 102: Bản đồ trạng thái - Khuấy nghịch Bồn 4 (State 23)
   RUNG wire#powerrail
      { S7_Templates := "SrcType := Int" } EQ_Contact(in1 := "PLC2_State", in2 := 23)
      Coil( "PLC2_Step_Bon4_Khuay_Nghich" )
   END_RUNG
   // the same network as SCL:
   "PLC2_Step_Bon4_Khuay_Nghich" := "PLC2_State" = 23;
END_REGION

REGION Network 103: Bản đồ trạng thái - PID Bồn 4 (State 30)
   RUNG wire#powerrail
      { S7_Templates := "SrcType := Int" } EQ_Contact(in1 := "PLC2_State", in2 := 30)
      Coil( "PLC2_Step_Bon4_PID_Mo_Phong" )
   END_RUNG
   // the same network as SCL:
   "PLC2_Step_Bon4_PID_Mo_Phong" := "PLC2_State" = 30;
END_REGION

REGION Network 104: Bản đồ trạng thái - Thanh trùng Bồn 4 (State 31)
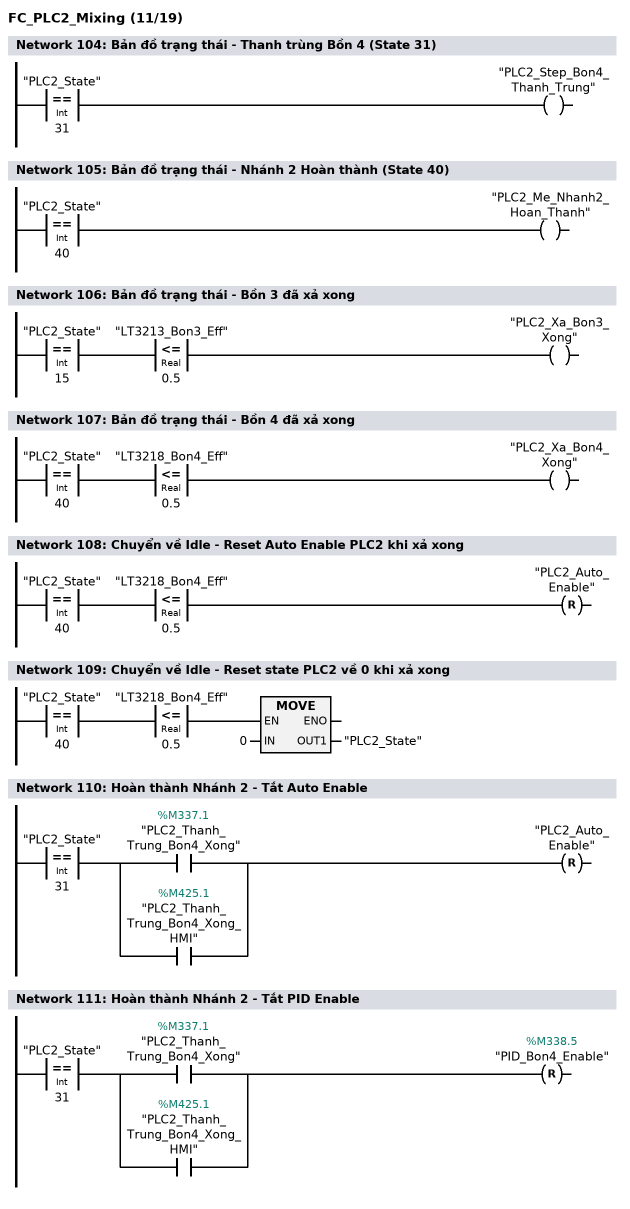
   RUNG wire#powerrail
      { S7_Templates := "SrcType := Int" } EQ_Contact(in1 := "PLC2_State", in2 := 31)
      Coil( "PLC2_Step_Bon4_Thanh_Trung" )
   END_RUNG
   // the same network as SCL:
   "PLC2_Step_Bon4_Thanh_Trung" := "PLC2_State" = 31;
END_REGION

REGION Network 105: Bản đồ trạng thái - Nhánh 2 Hoàn thành (State 40)
   RUNG wire#powerrail
      { S7_Templates := "SrcType := Int" } EQ_Contact(in1 := "PLC2_State", in2 := 40)
      Coil( "PLC2_Me_Nhanh2_Hoan_Thanh" )
   END_RUNG
   // the same network as SCL:
   "PLC2_Me_Nhanh2_Hoan_Thanh" := "PLC2_State" = 40;
END_REGION

REGION Network 106: Bản đồ trạng thái - Bồn 3 đã xả xong
   RUNG wire#powerrail
      { S7_Templates := "SrcType := Int" } EQ_Contact(in1 := "PLC2_State", in2 := 15)
      { S7_Templates := "SrcType := Real" } LE_Contact(in1 := "LT3213_Bon3_Eff", in2 := 0.5)
      Coil( "PLC2_Xa_Bon3_Xong" )
   END_RUNG
   // the same network as SCL:
   "PLC2_Xa_Bon3_Xong" := ("PLC2_State" = 15) AND ("LT3213_Bon3_Eff" <= 0.5);
END_REGION

REGION Network 107: Bản đồ trạng thái - Bồn 4 đã xả xong
   RUNG wire#powerrail
      { S7_Templates := "SrcType := Int" } EQ_Contact(in1 := "PLC2_State", in2 := 40)
      { S7_Templates := "SrcType := Real" } LE_Contact(in1 := "LT3218_Bon4_Eff", in2 := 0.5)
      Coil( "PLC2_Xa_Bon4_Xong" )
   END_RUNG
   // the same network as SCL:
   "PLC2_Xa_Bon4_Xong" := ("PLC2_State" = 40) AND ("LT3218_Bon4_Eff" <= 0.5);
END_REGION

REGION Network 108: Chuyển về Idle - Reset Auto Enable PLC2 khi xả xong
   RUNG wire#powerrail
      { S7_Templates := "SrcType := Int" } EQ_Contact(in1 := "PLC2_State", in2 := 40)
      { S7_Templates := "SrcType := Real" } LE_Contact(in1 := "LT3218_Bon4_Eff", in2 := 0.5)
      R_Coil( "PLC2_Auto_Enable" )
   END_RUNG
   // the same network as SCL:
   IF ("PLC2_State" = 40) AND ("LT3218_Bon4_Eff" <= 0.5) THEN "PLC2_Auto_Enable" := FALSE; END_IF;
END_REGION

REGION Network 109: Chuyển về Idle - Reset state PLC2 về 0 khi xả xong
   RUNG wire#powerrail
      { S7_Templates := "SrcType := Int" } EQ_Contact(in1 := "PLC2_State", in2 := 40)
      { S7_Templates := "SrcType := Real" } LE_Contact(in1 := "LT3218_Bon4_Eff", in2 := 0.5)
      { S7_GenerateENO := "TRUE" } Move(in := 0, out1 => "PLC2_State")
   END_RUNG
   // the same network as SCL:
   IF ("PLC2_State" = 40) AND ("LT3218_Bon4_Eff" <= 0.5) THEN "PLC2_State" := 0; END_IF;
END_REGION

REGION Network 110: Hoàn thành Nhánh 2 - Tắt Auto Enable
   RUNG wire#powerrail
      { S7_Templates := "SrcType := Int" } EQ_Contact(in1 := "PLC2_State", in2 := 31)
      wire#w1
      Contact( "PLC2_Thanh_Trung_Bon4_Xong" )
      wire#w2
      R_Coil( "PLC2_Auto_Enable" )
   END_RUNG
   RUNG wire#w1
      Contact( "PLC2_Thanh_Trung_Bon4_Xong_HMI" )
   END_RUNG wire#w2
   // the same network as SCL:
   IF ("PLC2_State" = 31) AND ("PLC2_Thanh_Trung_Bon4_Xong" OR "PLC2_Thanh_Trung_Bon4_Xong_HMI") THEN
       "PLC2_Auto_Enable" := FALSE;
   END_IF;
END_REGION

REGION Network 111: Hoàn thành Nhánh 2 - Tắt PID Enable
   RUNG wire#powerrail
      { S7_Templates := "SrcType := Int" } EQ_Contact(in1 := "PLC2_State", in2 := 31)
      wire#w1
      Contact( "PLC2_Thanh_Trung_Bon4_Xong" )
      wire#w2
      R_Coil( "PID_Bon4_Enable" )
   END_RUNG
   RUNG wire#w1
      Contact( "PLC2_Thanh_Trung_Bon4_Xong_HMI" )
   END_RUNG wire#w2
   // the same network as SCL:
   IF ("PLC2_State" = 31) AND ("PLC2_Thanh_Trung_Bon4_Xong" OR "PLC2_Thanh_Trung_Bon4_Xong_HMI") THEN
       "PID_Bon4_Enable" := FALSE;
   END_IF;
END_REGION

REGION Network 112: Hoàn thành Nhánh 2 - Chuyển sang State 40
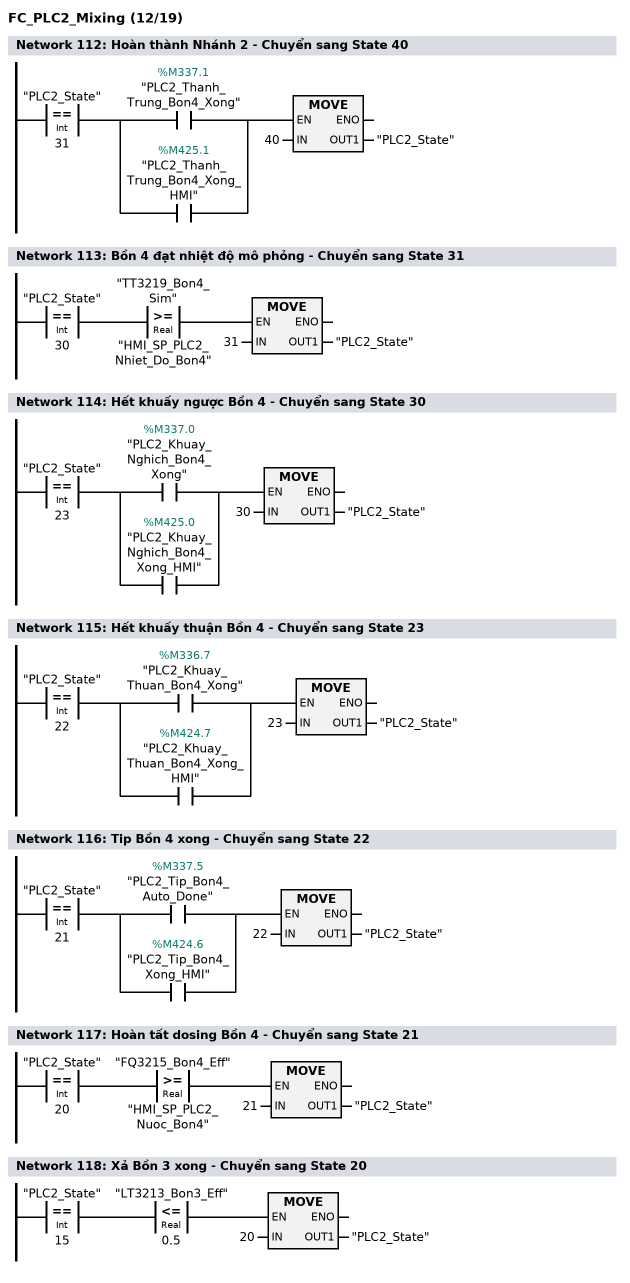
   RUNG wire#powerrail
      { S7_Templates := "SrcType := Int" } EQ_Contact(in1 := "PLC2_State", in2 := 31)
      wire#w1
      Contact( "PLC2_Thanh_Trung_Bon4_Xong" )
      wire#w2
      { S7_GenerateENO := "TRUE" } Move(in := 40, out1 => "PLC2_State")
   END_RUNG
   RUNG wire#w1
      Contact( "PLC2_Thanh_Trung_Bon4_Xong_HMI" )
   END_RUNG wire#w2
   // the same network as SCL:
   IF ("PLC2_State" = 31) AND ("PLC2_Thanh_Trung_Bon4_Xong" OR "PLC2_Thanh_Trung_Bon4_Xong_HMI") THEN
       "PLC2_State" := 40;
   END_IF;
END_REGION

REGION Network 113: Bồn 4 đạt nhiệt độ mô phỏng - Chuyển sang State 31
   RUNG wire#powerrail
      { S7_Templates := "SrcType := Int" } EQ_Contact(in1 := "PLC2_State", in2 := 30)
      { S7_Templates := "SrcType := Real" } GE_Contact(in1 := "TT3219_Bon4_Sim", in2 := "HMI_SP_PLC2_Nhiet_Do_Bon4")
      { S7_GenerateENO := "TRUE" } Move(in := 31, out1 => "PLC2_State")
   END_RUNG
   // the same network as SCL:
   IF ("PLC2_State" = 30) AND ("TT3219_Bon4_Sim" >= "HMI_SP_PLC2_Nhiet_Do_Bon4") THEN
       "PLC2_State" := 31;
   END_IF;
END_REGION

REGION Network 114: Hết khuấy ngược Bồn 4 - Chuyển sang State 30
   RUNG wire#powerrail
      { S7_Templates := "SrcType := Int" } EQ_Contact(in1 := "PLC2_State", in2 := 23)
      wire#w1
      Contact( "PLC2_Khuay_Nghich_Bon4_Xong" )
      wire#w2
      { S7_GenerateENO := "TRUE" } Move(in := 30, out1 => "PLC2_State")
   END_RUNG
   RUNG wire#w1
      Contact( "PLC2_Khuay_Nghich_Bon4_Xong_HMI" )
   END_RUNG wire#w2
   // the same network as SCL:
   IF ("PLC2_State" = 23) AND ("PLC2_Khuay_Nghich_Bon4_Xong" OR "PLC2_Khuay_Nghich_Bon4_Xong_HMI") THEN
       "PLC2_State" := 30;
   END_IF;
END_REGION

REGION Network 115: Hết khuấy thuận Bồn 4 - Chuyển sang State 23
   RUNG wire#powerrail
      { S7_Templates := "SrcType := Int" } EQ_Contact(in1 := "PLC2_State", in2 := 22)
      wire#w1
      Contact( "PLC2_Khuay_Thuan_Bon4_Xong" )
      wire#w2
      { S7_GenerateENO := "TRUE" } Move(in := 23, out1 => "PLC2_State")
   END_RUNG
   RUNG wire#w1
      Contact( "PLC2_Khuay_Thuan_Bon4_Xong_HMI" )
   END_RUNG wire#w2
   // the same network as SCL:
   IF ("PLC2_State" = 22) AND ("PLC2_Khuay_Thuan_Bon4_Xong" OR "PLC2_Khuay_Thuan_Bon4_Xong_HMI") THEN
       "PLC2_State" := 23;
   END_IF;
END_REGION

REGION Network 116: Tip Bồn 4 xong - Chuyển sang State 22
   RUNG wire#powerrail
      { S7_Templates := "SrcType := Int" } EQ_Contact(in1 := "PLC2_State", in2 := 21)
      wire#w1
      Contact( "PLC2_Tip_Bon4_Auto_Done" )
      wire#w2
      { S7_GenerateENO := "TRUE" } Move(in := 22, out1 => "PLC2_State")
   END_RUNG
   RUNG wire#w1
      Contact( "PLC2_Tip_Bon4_Xong_HMI" )
   END_RUNG wire#w2
   // the same network as SCL:
   IF ("PLC2_State" = 21) AND ("PLC2_Tip_Bon4_Auto_Done" OR "PLC2_Tip_Bon4_Xong_HMI") THEN
       "PLC2_State" := 22;
   END_IF;
END_REGION

REGION Network 117: Hoàn tất dosing Bồn 4 - Chuyển sang State 21
   RUNG wire#powerrail
      { S7_Templates := "SrcType := Int" } EQ_Contact(in1 := "PLC2_State", in2 := 20)
      { S7_Templates := "SrcType := Real" } GE_Contact(in1 := "FQ3215_Bon4_Eff", in2 := "HMI_SP_PLC2_Nuoc_Bon4")
      { S7_GenerateENO := "TRUE" } Move(in := 21, out1 => "PLC2_State")
   END_RUNG
   // the same network as SCL:
   IF ("PLC2_State" = 20) AND ("FQ3215_Bon4_Eff" >= "HMI_SP_PLC2_Nuoc_Bon4") THEN "PLC2_State" := 21; END_IF;
END_REGION

REGION Network 118: Xả Bồn 3 xong - Chuyển sang State 20
   RUNG wire#powerrail
      { S7_Templates := "SrcType := Int" } EQ_Contact(in1 := "PLC2_State", in2 := 15)
      { S7_Templates := "SrcType := Real" } LE_Contact(in1 := "LT3213_Bon3_Eff", in2 := 0.5)
      { S7_GenerateENO := "TRUE" } Move(in := 20, out1 => "PLC2_State")
   END_RUNG
   // the same network as SCL:
   IF ("PLC2_State" = 15) AND ("LT3213_Bon3_Eff" <= 0.5) THEN "PLC2_State" := 20; END_IF;
END_REGION

REGION Network 119: Khuấy Bồn 3 xong - Chuyển sang State 15
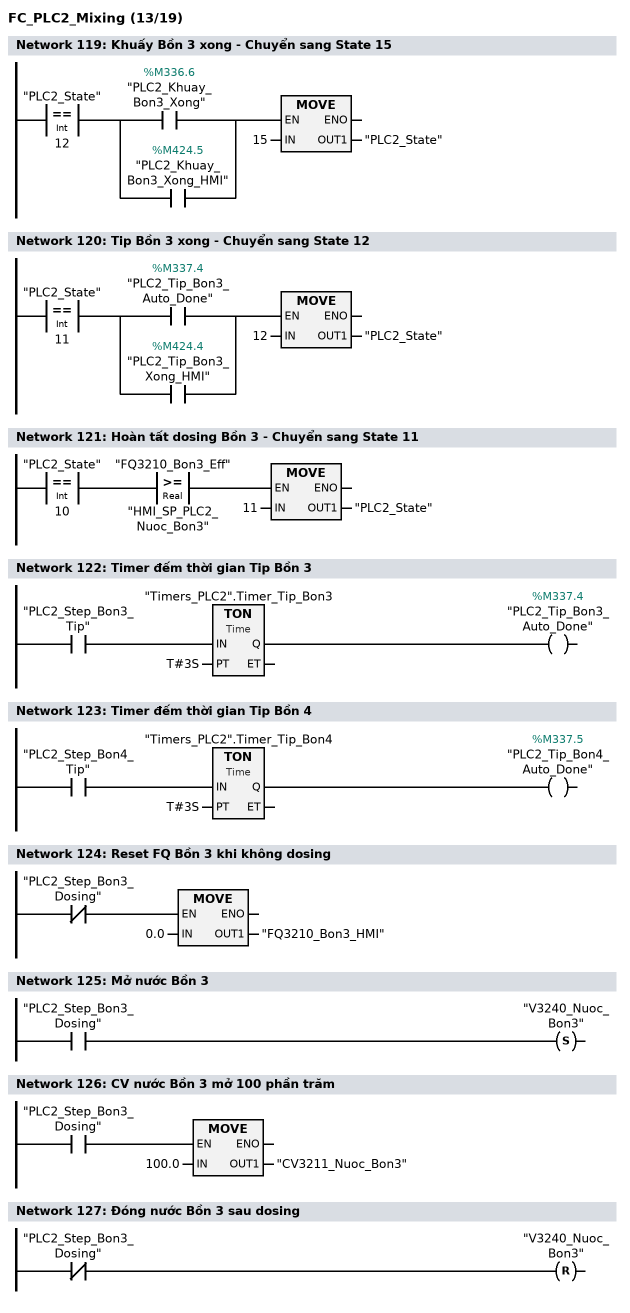
   RUNG wire#powerrail
      { S7_Templates := "SrcType := Int" } EQ_Contact(in1 := "PLC2_State", in2 := 12)
      wire#w1
      Contact( "PLC2_Khuay_Bon3_Xong" )
      wire#w2
      { S7_GenerateENO := "TRUE" } Move(in := 15, out1 => "PLC2_State")
   END_RUNG
   RUNG wire#w1
      Contact( "PLC2_Khuay_Bon3_Xong_HMI" )
   END_RUNG wire#w2
   // the same network as SCL:
   IF ("PLC2_State" = 12) AND ("PLC2_Khuay_Bon3_Xong" OR "PLC2_Khuay_Bon3_Xong_HMI") THEN
       "PLC2_State" := 15;
   END_IF;
END_REGION

REGION Network 120: Tip Bồn 3 xong - Chuyển sang State 12
   RUNG wire#powerrail
      { S7_Templates := "SrcType := Int" } EQ_Contact(in1 := "PLC2_State", in2 := 11)
      wire#w1
      Contact( "PLC2_Tip_Bon3_Auto_Done" )
      wire#w2
      { S7_GenerateENO := "TRUE" } Move(in := 12, out1 => "PLC2_State")
   END_RUNG
   RUNG wire#w1
      Contact( "PLC2_Tip_Bon3_Xong_HMI" )
   END_RUNG wire#w2
   // the same network as SCL:
   IF ("PLC2_State" = 11) AND ("PLC2_Tip_Bon3_Auto_Done" OR "PLC2_Tip_Bon3_Xong_HMI") THEN
       "PLC2_State" := 12;
   END_IF;
END_REGION

REGION Network 121: Hoàn tất dosing Bồn 3 - Chuyển sang State 11
   RUNG wire#powerrail
      { S7_Templates := "SrcType := Int" } EQ_Contact(in1 := "PLC2_State", in2 := 10)
      { S7_Templates := "SrcType := Real" } GE_Contact(in1 := "FQ3210_Bon3_Eff", in2 := "HMI_SP_PLC2_Nuoc_Bon3")
      { S7_GenerateENO := "TRUE" } Move(in := 11, out1 => "PLC2_State")
   END_RUNG
   // the same network as SCL:
   IF ("PLC2_State" = 10) AND ("FQ3210_Bon3_Eff" >= "HMI_SP_PLC2_Nuoc_Bon3") THEN "PLC2_State" := 11; END_IF;
END_REGION

REGION Network 122: Timer đếm thời gian Tip Bồn 3
   RUNG wire#powerrail
      Contact( "PLC2_Step_Bon3_Tip" )
      { S7_Templates := "time_type := Time" } "Timers_PLC2".Timer_Tip_Bon3.TON(pt := T#3S, et =>)
      Coil( "PLC2_Tip_Bon3_Auto_Done" )
   END_RUNG
   // the same network as SCL:
   "Timers_PLC2".Timer_Tip_Bon3.TON(IN := "PLC2_Step_Bon3_Tip", PT := T#3S);
   "PLC2_Tip_Bon3_Auto_Done" := "Timers_PLC2".Timer_Tip_Bon3.Q;
END_REGION

REGION Network 123: Timer đếm thời gian Tip Bồn 4
   RUNG wire#powerrail
      Contact( "PLC2_Step_Bon4_Tip" )
      { S7_Templates := "time_type := Time" } "Timers_PLC2".Timer_Tip_Bon4.TON(pt := T#3S, et =>)
      Coil( "PLC2_Tip_Bon4_Auto_Done" )
   END_RUNG
   // the same network as SCL:
   "Timers_PLC2".Timer_Tip_Bon4.TON(IN := "PLC2_Step_Bon4_Tip", PT := T#3S);
   "PLC2_Tip_Bon4_Auto_Done" := "Timers_PLC2".Timer_Tip_Bon4.Q;
END_REGION

REGION Network 124: Reset FQ Bồn 3 khi không dosing
   RUNG wire#powerrail
      I_Contact( "PLC2_Step_Bon3_Dosing" )
      { S7_GenerateENO := "TRUE" } Move(in := 0.0, out1 => "FQ3210_Bon3_HMI")
   END_RUNG
   // the same network as SCL:
   IF NOT "PLC2_Step_Bon3_Dosing" THEN "FQ3210_Bon3_HMI" := 0.0; END_IF;
END_REGION

REGION Network 125: Mở nước Bồn 3
   RUNG wire#powerrail
      Contact( "PLC2_Step_Bon3_Dosing" )
      S_Coil( "V3240_Nuoc_Bon3" )
   END_RUNG
   // the same network as SCL:
   IF "PLC2_Step_Bon3_Dosing" THEN "V3240_Nuoc_Bon3" := TRUE; END_IF;
END_REGION

REGION Network 126: CV nước Bồn 3 mở 100 phần trăm
   RUNG wire#powerrail
      Contact( "PLC2_Step_Bon3_Dosing" )
      { S7_GenerateENO := "TRUE" } Move(in := 100.0, out1 => "CV3211_Nuoc_Bon3")
   END_RUNG
   // the same network as SCL:
   IF "PLC2_Step_Bon3_Dosing" THEN "CV3211_Nuoc_Bon3" := 100.0; END_IF;
END_REGION

REGION Network 127: Đóng nước Bồn 3 sau dosing
   RUNG wire#powerrail
      I_Contact( "PLC2_Step_Bon3_Dosing" )
      R_Coil( "V3240_Nuoc_Bon3" )
   END_RUNG
   // the same network as SCL:
   IF NOT "PLC2_Step_Bon3_Dosing" THEN "V3240_Nuoc_Bon3" := FALSE; END_IF;
END_REGION

REGION Network 128: Đặt tốc độ khuấy Bồn 3
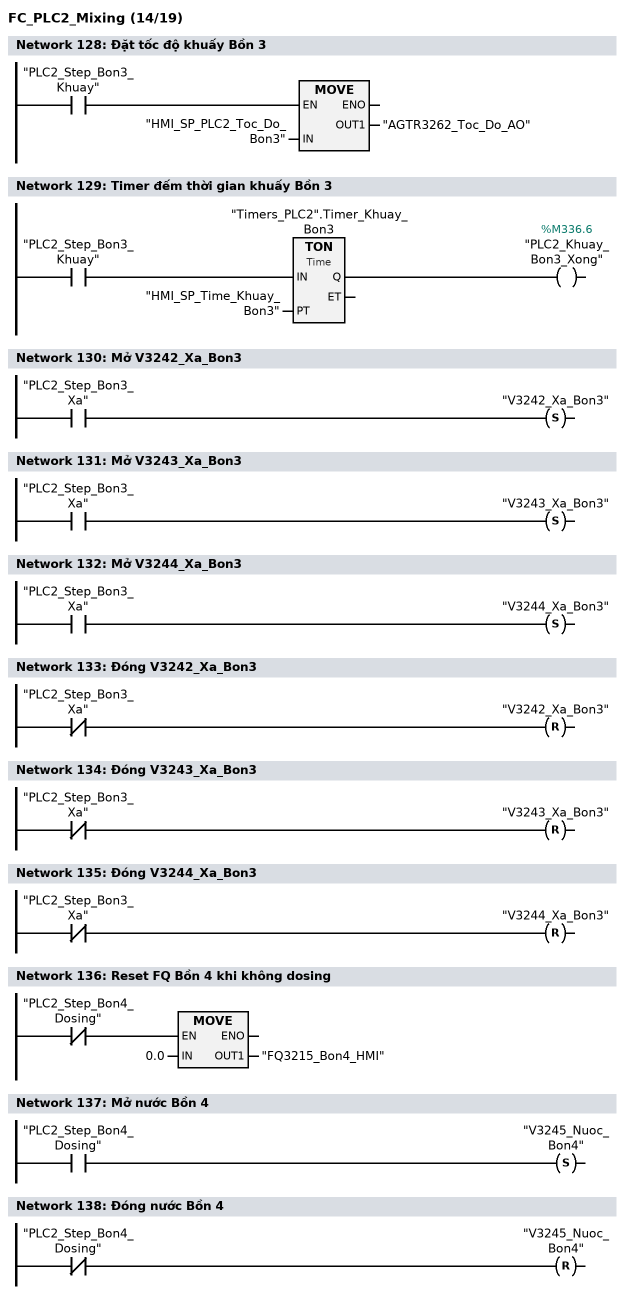
   RUNG wire#powerrail
      Contact( "PLC2_Step_Bon3_Khuay" )
      { S7_GenerateENO := "TRUE" } Move(in := "HMI_SP_PLC2_Toc_Do_Bon3", out1 => "AGTR3262_Toc_Do_AO")
   END_RUNG
   // the same network as SCL:
   IF "PLC2_Step_Bon3_Khuay" THEN "AGTR3262_Toc_Do_AO" := "HMI_SP_PLC2_Toc_Do_Bon3"; END_IF;
END_REGION

REGION Network 129: Timer đếm thời gian khuấy Bồn 3
   RUNG wire#powerrail
      Contact( "PLC2_Step_Bon3_Khuay" )
      { S7_Templates := "time_type := Time" } "Timers_PLC2".Timer_Khuay_Bon3.TON(pt := "HMI_SP_Time_Khuay_Bon3", et =>)
      Coil( "PLC2_Khuay_Bon3_Xong" )
   END_RUNG
   // the same network as SCL:
   "Timers_PLC2".Timer_Khuay_Bon3.TON(IN := "PLC2_Step_Bon3_Khuay", PT := "HMI_SP_Time_Khuay_Bon3");
   "PLC2_Khuay_Bon3_Xong" := "Timers_PLC2".Timer_Khuay_Bon3.Q;
END_REGION

REGION Network 130: Mở V3242_Xa_Bon3
   RUNG wire#powerrail
      Contact( "PLC2_Step_Bon3_Xa" )
      S_Coil( "V3242_Xa_Bon3" )
   END_RUNG
   // the same network as SCL:
   IF "PLC2_Step_Bon3_Xa" THEN "V3242_Xa_Bon3" := TRUE; END_IF;
END_REGION

REGION Network 131: Mở V3243_Xa_Bon3
   RUNG wire#powerrail
      Contact( "PLC2_Step_Bon3_Xa" )
      S_Coil( "V3243_Xa_Bon3" )
   END_RUNG
   // the same network as SCL:
   IF "PLC2_Step_Bon3_Xa" THEN "V3243_Xa_Bon3" := TRUE; END_IF;
END_REGION

REGION Network 132: Mở V3244_Xa_Bon3
   RUNG wire#powerrail
      Contact( "PLC2_Step_Bon3_Xa" )
      S_Coil( "V3244_Xa_Bon3" )
   END_RUNG
   // the same network as SCL:
   IF "PLC2_Step_Bon3_Xa" THEN "V3244_Xa_Bon3" := TRUE; END_IF;
END_REGION

REGION Network 133: Đóng V3242_Xa_Bon3
   RUNG wire#powerrail
      I_Contact( "PLC2_Step_Bon3_Xa" )
      R_Coil( "V3242_Xa_Bon3" )
   END_RUNG
   // the same network as SCL:
   IF NOT "PLC2_Step_Bon3_Xa" THEN "V3242_Xa_Bon3" := FALSE; END_IF;
END_REGION

REGION Network 134: Đóng V3243_Xa_Bon3
   RUNG wire#powerrail
      I_Contact( "PLC2_Step_Bon3_Xa" )
      R_Coil( "V3243_Xa_Bon3" )
   END_RUNG
   // the same network as SCL:
   IF NOT "PLC2_Step_Bon3_Xa" THEN "V3243_Xa_Bon3" := FALSE; END_IF;
END_REGION

REGION Network 135: Đóng V3244_Xa_Bon3
   RUNG wire#powerrail
      I_Contact( "PLC2_Step_Bon3_Xa" )
      R_Coil( "V3244_Xa_Bon3" )
   END_RUNG
   // the same network as SCL:
   IF NOT "PLC2_Step_Bon3_Xa" THEN "V3244_Xa_Bon3" := FALSE; END_IF;
END_REGION

REGION Network 136: Reset FQ Bồn 4 khi không dosing
   RUNG wire#powerrail
      I_Contact( "PLC2_Step_Bon4_Dosing" )
      { S7_GenerateENO := "TRUE" } Move(in := 0.0, out1 => "FQ3215_Bon4_HMI")
   END_RUNG
   // the same network as SCL:
   IF NOT "PLC2_Step_Bon4_Dosing" THEN "FQ3215_Bon4_HMI" := 0.0; END_IF;
END_REGION

REGION Network 137: Mở nước Bồn 4
   RUNG wire#powerrail
      Contact( "PLC2_Step_Bon4_Dosing" )
      S_Coil( "V3245_Nuoc_Bon4" )
   END_RUNG
   // the same network as SCL:
   IF "PLC2_Step_Bon4_Dosing" THEN "V3245_Nuoc_Bon4" := TRUE; END_IF;
END_REGION

REGION Network 138: Đóng nước Bồn 4
   RUNG wire#powerrail
      I_Contact( "PLC2_Step_Bon4_Dosing" )
      R_Coil( "V3245_Nuoc_Bon4" )
   END_RUNG
   // the same network as SCL:
   IF NOT "PLC2_Step_Bon4_Dosing" THEN "V3245_Nuoc_Bon4" := FALSE; END_IF;
END_REGION

REGION Network 139: Tốc độ khuấy thuận Bồn 4
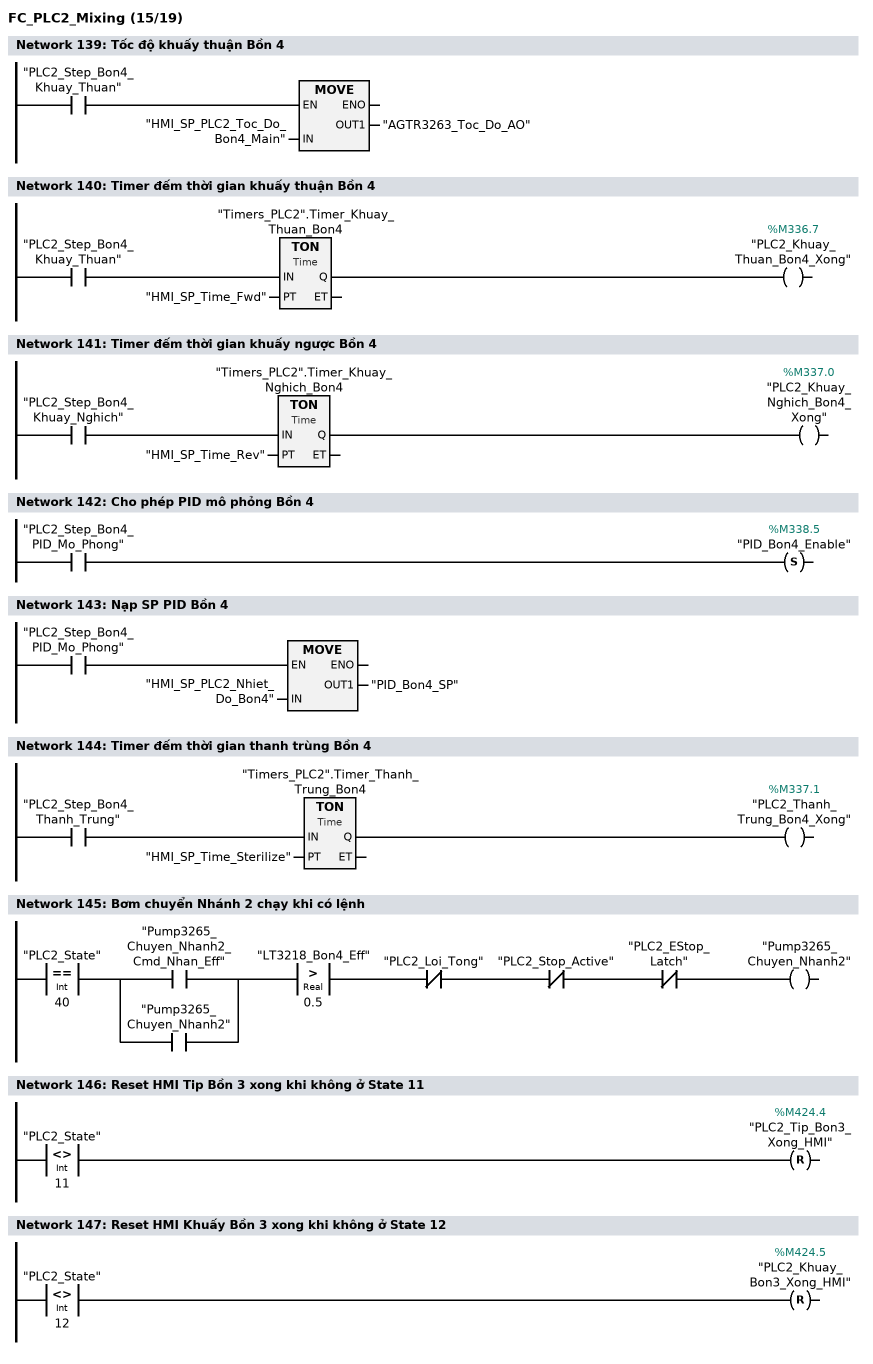
   RUNG wire#powerrail
      Contact( "PLC2_Step_Bon4_Khuay_Thuan" )
      { S7_GenerateENO := "TRUE" } Move(in := "HMI_SP_PLC2_Toc_Do_Bon4_Main", out1 => "AGTR3263_Toc_Do_AO")
   END_RUNG
   // the same network as SCL:
   IF "PLC2_Step_Bon4_Khuay_Thuan" THEN "AGTR3263_Toc_Do_AO" := "HMI_SP_PLC2_Toc_Do_Bon4_Main"; END_IF;
END_REGION

REGION Network 140: Timer đếm thời gian khuấy thuận Bồn 4
   RUNG wire#powerrail
      Contact( "PLC2_Step_Bon4_Khuay_Thuan" )
      { S7_Templates := "time_type := Time" } "Timers_PLC2".Timer_Khuay_Thuan_Bon4.TON(pt := "HMI_SP_Time_Fwd", et =>)
      Coil( "PLC2_Khuay_Thuan_Bon4_Xong" )
   END_RUNG
   // the same network as SCL:
   "Timers_PLC2".Timer_Khuay_Thuan_Bon4.TON(IN := "PLC2_Step_Bon4_Khuay_Thuan", PT := "HMI_SP_Time_Fwd");
   "PLC2_Khuay_Thuan_Bon4_Xong" := "Timers_PLC2".Timer_Khuay_Thuan_Bon4.Q;
END_REGION

REGION Network 141: Timer đếm thời gian khuấy ngược Bồn 4
   RUNG wire#powerrail
      Contact( "PLC2_Step_Bon4_Khuay_Nghich" )
      { S7_Templates := "time_type := Time" } "Timers_PLC2".Timer_Khuay_Nghich_Bon4.TON(pt := "HMI_SP_Time_Rev", et =>)
      Coil( "PLC2_Khuay_Nghich_Bon4_Xong" )
   END_RUNG
   // the same network as SCL:
   "Timers_PLC2".Timer_Khuay_Nghich_Bon4.TON(IN := "PLC2_Step_Bon4_Khuay_Nghich", PT := "HMI_SP_Time_Rev");
   "PLC2_Khuay_Nghich_Bon4_Xong" := "Timers_PLC2".Timer_Khuay_Nghich_Bon4.Q;
END_REGION

REGION Network 142: Cho phép PID mô phỏng Bồn 4
   RUNG wire#powerrail
      Contact( "PLC2_Step_Bon4_PID_Mo_Phong" )
      S_Coil( "PID_Bon4_Enable" )
   END_RUNG
   // the same network as SCL:
   IF "PLC2_Step_Bon4_PID_Mo_Phong" THEN "PID_Bon4_Enable" := TRUE; END_IF;
END_REGION

REGION Network 143: Nạp SP PID Bồn 4
   RUNG wire#powerrail
      Contact( "PLC2_Step_Bon4_PID_Mo_Phong" )
      { S7_GenerateENO := "TRUE" } Move(in := "HMI_SP_PLC2_Nhiet_Do_Bon4", out1 => "PID_Bon4_SP")
   END_RUNG
   // the same network as SCL:
   IF "PLC2_Step_Bon4_PID_Mo_Phong" THEN "PID_Bon4_SP" := "HMI_SP_PLC2_Nhiet_Do_Bon4"; END_IF;
END_REGION

REGION Network 144: Timer đếm thời gian thanh trùng Bồn 4
   RUNG wire#powerrail
      Contact( "PLC2_Step_Bon4_Thanh_Trung" )
      { S7_Templates := "time_type := Time" } "Timers_PLC2".Timer_Thanh_Trung_Bon4.TON(pt := "HMI_SP_Time_Sterilize", et =>)
      Coil( "PLC2_Thanh_Trung_Bon4_Xong" )
   END_RUNG
   // the same network as SCL:
   "Timers_PLC2".Timer_Thanh_Trung_Bon4.TON(IN := "PLC2_Step_Bon4_Thanh_Trung", PT := "HMI_SP_Time_Sterilize");
   "PLC2_Thanh_Trung_Bon4_Xong" := "Timers_PLC2".Timer_Thanh_Trung_Bon4.Q;
END_REGION

REGION Network 145: Bơm chuyển Nhánh 2 chạy khi có lệnh
   RUNG wire#powerrail
      { S7_Templates := "SrcType := Int" } EQ_Contact(in1 := "PLC2_State", in2 := 40)
      wire#w1
      Contact( "Pump3265_Chuyen_Nhanh2_Cmd_Nhan_Eff" )
      wire#w2
      { S7_Templates := "SrcType := Real" } GT_Contact(in1 := "LT3218_Bon4_Eff", in2 := 0.5)
      I_Contact( "PLC2_Loi_Tong" )
      I_Contact( "PLC2_Stop_Active" )
      I_Contact( "PLC2_EStop_Latch" )
      Coil( "Pump3265_Chuyen_Nhanh2" )
   END_RUNG
   RUNG wire#w1
      Contact( "Pump3265_Chuyen_Nhanh2" )
   END_RUNG wire#w2
   // the same network as SCL:
   "Pump3265_Chuyen_Nhanh2" := ("PLC2_State" = 40) AND ("Pump3265_Chuyen_Nhanh2_Cmd_Nhan_Eff" OR "Pump3265_Chuyen_Nhanh2") AND ("LT3218_Bon4_Eff" > 0.5) AND NOT "PLC2_Loi_Tong" AND NOT "PLC2_Stop_Active" AND NOT "PLC2_EStop_Latch";
END_REGION

REGION Network 146: Reset HMI Tip Bồn 3 xong khi không ở State 11
   RUNG wire#powerrail
      { S7_Templates := "SrcType := Int" } NE_Contact(in1 := "PLC2_State", in2 := 11)
      R_Coil( "PLC2_Tip_Bon3_Xong_HMI" )
   END_RUNG
   // the same network as SCL:
   IF "PLC2_State" <> 11 THEN "PLC2_Tip_Bon3_Xong_HMI" := FALSE; END_IF;
END_REGION

REGION Network 147: Reset HMI Khuấy Bồn 3 xong khi không ở State 12
   RUNG wire#powerrail
      { S7_Templates := "SrcType := Int" } NE_Contact(in1 := "PLC2_State", in2 := 12)
      R_Coil( "PLC2_Khuay_Bon3_Xong_HMI" )
   END_RUNG
   // the same network as SCL:
   IF "PLC2_State" <> 12 THEN "PLC2_Khuay_Bon3_Xong_HMI" := FALSE; END_IF;
END_REGION

REGION Network 148: Reset HMI Tip Bồn 4 xong khi không ở State 21
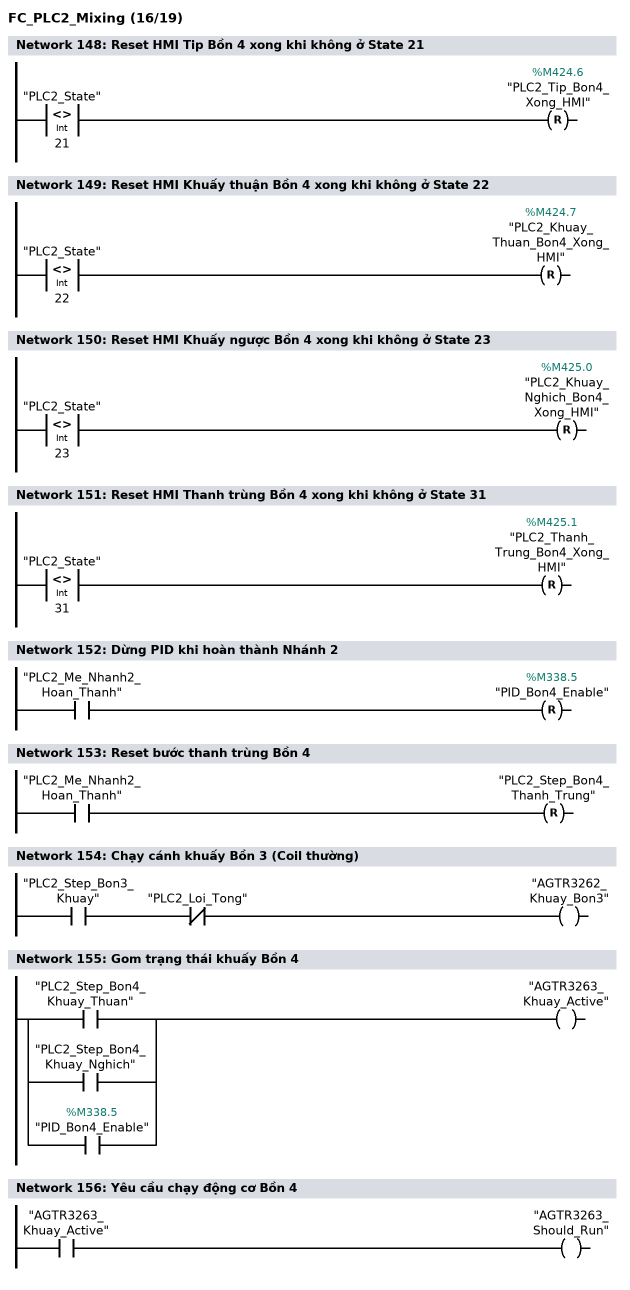
   RUNG wire#powerrail
      { S7_Templates := "SrcType := Int" } NE_Contact(in1 := "PLC2_State", in2 := 21)
      R_Coil( "PLC2_Tip_Bon4_Xong_HMI" )
   END_RUNG
   // the same network as SCL:
   IF "PLC2_State" <> 21 THEN "PLC2_Tip_Bon4_Xong_HMI" := FALSE; END_IF;
END_REGION

REGION Network 149: Reset HMI Khuấy thuận Bồn 4 xong khi không ở State 22
   RUNG wire#powerrail
      { S7_Templates := "SrcType := Int" } NE_Contact(in1 := "PLC2_State", in2 := 22)
      R_Coil( "PLC2_Khuay_Thuan_Bon4_Xong_HMI" )
   END_RUNG
   // the same network as SCL:
   IF "PLC2_State" <> 22 THEN "PLC2_Khuay_Thuan_Bon4_Xong_HMI" := FALSE; END_IF;
END_REGION

REGION Network 150: Reset HMI Khuấy ngược Bồn 4 xong khi không ở State 23
   RUNG wire#powerrail
      { S7_Templates := "SrcType := Int" } NE_Contact(in1 := "PLC2_State", in2 := 23)
      R_Coil( "PLC2_Khuay_Nghich_Bon4_Xong_HMI" )
   END_RUNG
   // the same network as SCL:
   IF "PLC2_State" <> 23 THEN "PLC2_Khuay_Nghich_Bon4_Xong_HMI" := FALSE; END_IF;
END_REGION

REGION Network 151: Reset HMI Thanh trùng Bồn 4 xong khi không ở State 31
   RUNG wire#powerrail
      { S7_Templates := "SrcType := Int" } NE_Contact(in1 := "PLC2_State", in2 := 31)
      R_Coil( "PLC2_Thanh_Trung_Bon4_Xong_HMI" )
   END_RUNG
   // the same network as SCL:
   IF "PLC2_State" <> 31 THEN "PLC2_Thanh_Trung_Bon4_Xong_HMI" := FALSE; END_IF;
END_REGION

REGION Network 152: Dừng PID khi hoàn thành Nhánh 2
   RUNG wire#powerrail
      Contact( "PLC2_Me_Nhanh2_Hoan_Thanh" )
      R_Coil( "PID_Bon4_Enable" )
   END_RUNG
   // the same network as SCL:
   IF "PLC2_Me_Nhanh2_Hoan_Thanh" THEN "PID_Bon4_Enable" := FALSE; END_IF;
END_REGION

REGION Network 153: Reset bước thanh trùng Bồn 4
   RUNG wire#powerrail
      Contact( "PLC2_Me_Nhanh2_Hoan_Thanh" )
      R_Coil( "PLC2_Step_Bon4_Thanh_Trung" )
   END_RUNG
   // the same network as SCL:
   IF "PLC2_Me_Nhanh2_Hoan_Thanh" THEN "PLC2_Step_Bon4_Thanh_Trung" := FALSE; END_IF;
END_REGION

REGION Network 154: Chạy cánh khuấy Bồn 3 (Coil thường)
   RUNG wire#powerrail
      Contact( "PLC2_Step_Bon3_Khuay" )
      I_Contact( "PLC2_Loi_Tong" )
      Coil( "AGTR3262_Khuay_Bon3" )
   END_RUNG
   // the same network as SCL:
   "AGTR3262_Khuay_Bon3" := "PLC2_Step_Bon3_Khuay" AND NOT "PLC2_Loi_Tong";
END_REGION

REGION Network 155: Gom trạng thái khuấy Bồn 4
   RUNG wire#powerrail
      Contact( "PLC2_Step_Bon4_Khuay_Thuan" )
      wire#w1
      Coil( "AGTR3263_Khuay_Active" )
   END_RUNG
   RUNG wire#powerrail
      Contact( "PLC2_Step_Bon4_Khuay_Nghich" )
   END_RUNG wire#w1
   RUNG wire#powerrail
      Contact( "PID_Bon4_Enable" )
   END_RUNG wire#w1
   // the same network as SCL:
   "AGTR3263_Khuay_Active" := "PLC2_Step_Bon4_Khuay_Thuan" OR "PLC2_Step_Bon4_Khuay_Nghich" OR "PID_Bon4_Enable";
END_REGION

REGION Network 156: Yêu cầu chạy động cơ Bồn 4
   RUNG wire#powerrail
      Contact( "AGTR3263_Khuay_Active" )
      Coil( "AGTR3263_Should_Run" )
   END_RUNG
   // the same network as SCL:
   "AGTR3263_Should_Run" := "AGTR3263_Khuay_Active";
END_REGION

REGION Network 157: Lệnh chạy động cơ khuấy Bồn 4 (Coil thường)
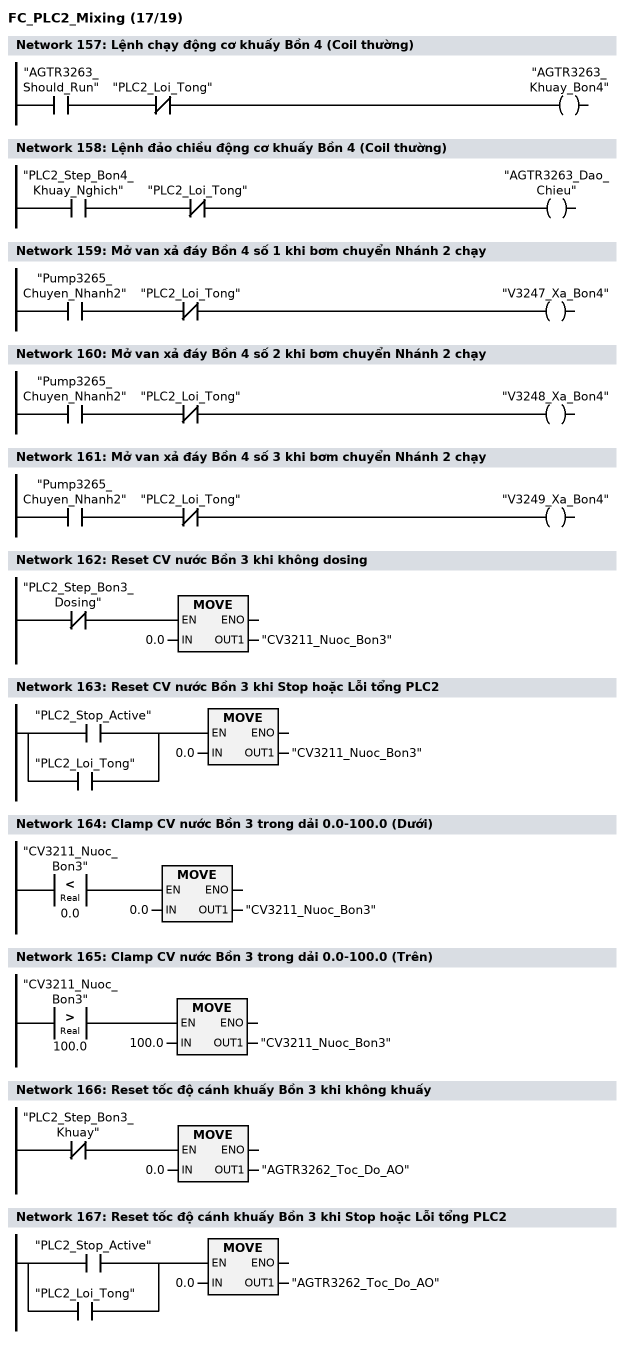
   RUNG wire#powerrail
      Contact( "AGTR3263_Should_Run" )
      I_Contact( "PLC2_Loi_Tong" )
      Coil( "AGTR3263_Khuay_Bon4" )
   END_RUNG
   // the same network as SCL:
   "AGTR3263_Khuay_Bon4" := "AGTR3263_Should_Run" AND NOT "PLC2_Loi_Tong";
END_REGION

REGION Network 158: Lệnh đảo chiều động cơ khuấy Bồn 4 (Coil thường)
   RUNG wire#powerrail
      Contact( "PLC2_Step_Bon4_Khuay_Nghich" )
      I_Contact( "PLC2_Loi_Tong" )
      Coil( "AGTR3263_Dao_Chieu" )
   END_RUNG
   // the same network as SCL:
   "AGTR3263_Dao_Chieu" := "PLC2_Step_Bon4_Khuay_Nghich" AND NOT "PLC2_Loi_Tong";
END_REGION

REGION Network 159: Mở van xả đáy Bồn 4 số 1 khi bơm chuyển Nhánh 2 chạy
   RUNG wire#powerrail
      Contact( "Pump3265_Chuyen_Nhanh2" )
      I_Contact( "PLC2_Loi_Tong" )
      Coil( "V3247_Xa_Bon4" )
   END_RUNG
   // the same network as SCL:
   "V3247_Xa_Bon4" := "Pump3265_Chuyen_Nhanh2" AND NOT "PLC2_Loi_Tong";
END_REGION

REGION Network 160: Mở van xả đáy Bồn 4 số 2 khi bơm chuyển Nhánh 2 chạy
   RUNG wire#powerrail
      Contact( "Pump3265_Chuyen_Nhanh2" )
      I_Contact( "PLC2_Loi_Tong" )
      Coil( "V3248_Xa_Bon4" )
   END_RUNG
   // the same network as SCL:
   "V3248_Xa_Bon4" := "Pump3265_Chuyen_Nhanh2" AND NOT "PLC2_Loi_Tong";
END_REGION

REGION Network 161: Mở van xả đáy Bồn 4 số 3 khi bơm chuyển Nhánh 2 chạy
   RUNG wire#powerrail
      Contact( "Pump3265_Chuyen_Nhanh2" )
      I_Contact( "PLC2_Loi_Tong" )
      Coil( "V3249_Xa_Bon4" )
   END_RUNG
   // the same network as SCL:
   "V3249_Xa_Bon4" := "Pump3265_Chuyen_Nhanh2" AND NOT "PLC2_Loi_Tong";
END_REGION

REGION Network 162: Reset CV nước Bồn 3 khi không dosing
   RUNG wire#powerrail
      I_Contact( "PLC2_Step_Bon3_Dosing" )
      { S7_GenerateENO := "TRUE" } Move(in := 0.0, out1 => "CV3211_Nuoc_Bon3")
   END_RUNG
   // the same network as SCL:
   IF NOT "PLC2_Step_Bon3_Dosing" THEN "CV3211_Nuoc_Bon3" := 0.0; END_IF;
END_REGION

REGION Network 163: Reset CV nước Bồn 3 khi Stop hoặc Lỗi tổng PLC2
   RUNG wire#powerrail
      Contact( "PLC2_Stop_Active" )
      wire#w1
      { S7_GenerateENO := "TRUE" } Move(in := 0.0, out1 => "CV3211_Nuoc_Bon3")
   END_RUNG
   RUNG wire#powerrail
      Contact( "PLC2_Loi_Tong" )
   END_RUNG wire#w1
   // the same network as SCL:
   IF "PLC2_Stop_Active" OR "PLC2_Loi_Tong" THEN "CV3211_Nuoc_Bon3" := 0.0; END_IF;
END_REGION

REGION Network 164: Clamp CV nước Bồn 3 trong dải 0.0-100.0 (Dưới)
   RUNG wire#powerrail
      { S7_Templates := "SrcType := Real" } LT_Contact(in1 := "CV3211_Nuoc_Bon3", in2 := 0.0)
      { S7_GenerateENO := "TRUE" } Move(in := 0.0, out1 => "CV3211_Nuoc_Bon3")
   END_RUNG
   // the same network as SCL:
   IF "CV3211_Nuoc_Bon3" < 0.0 THEN "CV3211_Nuoc_Bon3" := 0.0; END_IF;
END_REGION

REGION Network 165: Clamp CV nước Bồn 3 trong dải 0.0-100.0 (Trên)
   RUNG wire#powerrail
      { S7_Templates := "SrcType := Real" } GT_Contact(in1 := "CV3211_Nuoc_Bon3", in2 := 100.0)
      { S7_GenerateENO := "TRUE" } Move(in := 100.0, out1 => "CV3211_Nuoc_Bon3")
   END_RUNG
   // the same network as SCL:
   IF "CV3211_Nuoc_Bon3" > 100.0 THEN "CV3211_Nuoc_Bon3" := 100.0; END_IF;
END_REGION

REGION Network 166: Reset tốc độ cánh khuấy Bồn 3 khi không khuấy
   RUNG wire#powerrail
      I_Contact( "PLC2_Step_Bon3_Khuay" )
      { S7_GenerateENO := "TRUE" } Move(in := 0.0, out1 => "AGTR3262_Toc_Do_AO")
   END_RUNG
   // the same network as SCL:
   IF NOT "PLC2_Step_Bon3_Khuay" THEN "AGTR3262_Toc_Do_AO" := 0.0; END_IF;
END_REGION

REGION Network 167: Reset tốc độ cánh khuấy Bồn 3 khi Stop hoặc Lỗi tổng PLC2
   RUNG wire#powerrail
      Contact( "PLC2_Stop_Active" )
      wire#w1
      { S7_GenerateENO := "TRUE" } Move(in := 0.0, out1 => "AGTR3262_Toc_Do_AO")
   END_RUNG
   RUNG wire#powerrail
      Contact( "PLC2_Loi_Tong" )
   END_RUNG wire#w1
   // the same network as SCL:
   IF "PLC2_Stop_Active" OR "PLC2_Loi_Tong" THEN "AGTR3262_Toc_Do_AO" := 0.0; END_IF;
END_REGION

REGION Network 168: Clamp tốc độ cánh khuấy Bồn 3 trong dải 0.0-100.0 (Dưới)
